  MoveL 3801 to (497.52, 492.57, 7.8) mm, rotated rx 0 ry 90 rz 0 deg; joints [-11.373, -27.183, 111.629, -15.362, -83.781, 50.697]
  MoveL 3802 to (497.65, 492.45, 7.8) mm, rotated rx 0 ry 90 rz 0 deg; joints [-11.359, -27.181, 111.617, -15.349, -83.771, 50.699]
  Set speed (120.0 mm/s)
  MoveL 3803 to (502.42, 492.52, 7.8) mm, rotated rx 0 ry 90 rz 0 deg; joints [-11.277, -27.097, 111.047, -15.281, -83.3, 50.82]
  Set speed (30.0 mm/s)
  Call Extruder(0.230)
  MoveL 3804 to (508, 498.1, 7.8) mm, rotated rx 0 ry 90 rz 0 deg; joints [-11.683, -26.971, 110.241, -15.712, -82.657, 51.047]
  MoveL 3805 to (508.13, 498.23, 7.8) mm, rotated rx 0 ry 90 rz 0 deg; joints [-11.692, -26.968, 110.224, -15.722, -82.643, 51.052]
  Set speed (120.0 mm/s)
  MoveL 3806 to (509.32, 490.68, 7.8) mm, rotated rx 0 ry 90 rz 0 deg; joints [-10.985, -26.974, 110.262, -15.009, -82.652, 50.963]
  Set speed (30.0 mm/s)
  Call Extruder(0.767)
  MoveL 3807 to (490.68, 509.32, 7.8) mm, rotated rx 0 ry 90 rz 0 deg; joints [-13.056, -27.238, 112.01, -17.045, -84.139, 50.759]
  MoveL 3808 to (490.56, 509.44, 7.8) mm, rotated rx 0 ry 90 rz 0 deg; joints [-13.07, -27.239, 112.021, -17.059, -84.148, 50.757]
  Set speed (120.0 mm/s)
  MoveL 3809 to (499.58, 492.37, 7.8) mm, rotated rx 0 ry 90 rz 0 deg; joints [-11.315, -27.148, 111.389, -15.311, -83.582, 50.746]
  Set speed (1000.0 mm/s)
  MoveL 3810 to (499.65, 492.3, 7.8) mm, rotated rx 0 ry 90 rz 0 deg; joints [-11.307, -27.147, 111.382, -15.303, -83.576, 50.747]
  Set speed (15.0 mm/s)
  Call Extruder(0.010)
  MoveL 3811 to (500, 492.3, 7.8) mm, rotated rx 0 ry 90 rz 0 deg; joints [-11.301, -27.141, 111.341, -15.297, -83.542, 50.756]
  Call Extruder(0.000)
  MoveL 3812 to (500, 492.3, 7.8) mm, rotated rx 0 ry 90 rz 0 deg; joints [-11.301, -27.141, 111.34, -15.297, -83.542, 50.756]
  Call Extruder(0.062)
  MoveL 3813 to (502.14, 492.3, 7.8) mm, rotated rx 0 ry 90 rz 0 deg; joints [-11.262, -27.102, 111.085, -15.265, -83.331, 50.81]
  Call Extruder(0.055)
  MoveL 3814 to (502.14, 490.4, 7.8) mm, rotated rx 0 ry 90 rz 0 deg; joints [-11.088, -27.109, 111.13, -15.088, -83.363, 50.782]
  Call Extruder(0.217)
  MoveL 3815 to (509.6, 490.4, 7.8) mm, rotated rx 0 ry 90 rz 0 deg; joints [-10.955, -26.97, 110.235, -14.979, -82.629, 50.965]
  Call Extruder(0.232)
  MoveL 3816 to (509.6, 498.38, 7.8) mm, rotated rx 0 ry 90 rz 0 deg; joints [-11.678, -26.939, 110.042, -15.714, -82.496, 51.092]
  Call Extruder(0.046)
  MoveL 3817 to (508.01, 498.39, 7.8) mm, rotated rx 0 ry 90 rz 0 deg; joints [-11.708, -26.97, 110.233, -15.738, -82.651, 51.051]
  Call Extruder(0.010)
  MoveL 3818 to (507.66, 498.38, 7.8) mm, rotated rx 0 ry 90 rz 0 deg; joints [-11.715, -26.977, 110.275, -15.743, -82.686, 51.043]
  Call Extruder(0.007)
  MoveL 3819 to (507.66, 498.74, 7.8) mm, rotated rx 0 ry 90 rz 0 deg; joints [-11.746, -26.975, 110.267, -15.776, -82.68, 51.048]
  Call Extruder(0.062)
  MoveL 3820 to (507.66, 500.87, 7.8) mm, rotated rx 0 ry 90 rz 0 deg; joints [-11.939, -26.967, 110.213, -15.971, -82.642, 51.083]
  Call Extruder(0.056)
  MoveL 3821 to (509.6, 500.87, 7.8) mm, rotated rx 0 ry 90 rz 0 deg; joints [-11.902, -26.929, 109.98, -15.941, -82.453, 51.132]
  Call Extruder(0.254)
  MoveL 3822 to (509.6, 509.6, 7.8) mm, rotated rx 0 ry 90 rz 0 deg; joints [-12.688, -26.891, 109.751, -16.741, -82.297, 51.28]
  Call Extruder(0.559)
  MoveL 3823 to (490.4, 509.6, 7.8) mm, rotated rx 0 ry 90 rz 0 deg; joints [-13.088, -27.241, 112.035, -17.076, -84.16, 50.755]
  MoveL 3824 to (490.4, 490.4, 7.8) mm, rotated rx 0 ry 90 rz 0 deg; joints [-11.303, -27.309, 112.525, -15.272, -84.522, 50.487]
  Call Extruder(0.189)
  MoveL 3825 to (496.9, 490.4, 7.8) mm, rotated rx 0 ry 90 rz 0 deg; joints [-11.183, -27.201, 111.755, -15.169, -83.88, 50.651]
  Call Extruder(0.055)
  MoveL 3826 to (496.9, 492.3, 7.8) mm, rotated rx 0 ry 90 rz 0 deg; joints [-11.358, -27.195, 111.71, -15.346, -83.847, 50.678]
  Call Extruder(0.075)
  MoveL 3827 to (499.46, 492.29, 7.8) mm, rotated rx 0 ry 90 rz 0 deg; joints [-11.311, -27.15, 111.405, -15.306, -83.595, 50.742]
  Call Extruder(0.021)
  MoveL 3828 to (499.46, 491.57, 7.8) mm, rotated rx 0 ry 90 rz 0 deg; joints [-11.244, -27.153, 111.422, -15.238, -83.607, 50.732]
  Call Extruder(0.034)
  MoveL 3829 to (499.46, 490.4, 7.8) mm, rotated rx 0 ry 90 rz 0 deg; joints [-11.136, -27.157, 111.45, -15.129, -83.627, 50.715]
  Call Extruder(0.006)
  MoveL 3830 to (499.66, 490.4, 7.8) mm, rotated rx 0 ry 90 rz 0 deg; joints [-11.133, -27.154, 111.427, -15.126, -83.608, 50.72]
  Call Extruder(0.009)
  MoveL 3831 to (499.66, 491.57, 7.8) mm, rotated rx 0 ry 90 rz 0 deg; joints [-11.241, -27.149, 111.399, -15.235, -83.588, 50.737]
  Call Extruder(0.011)
  MoveL 3832 to (499.65, 491.94, 7.8) mm, rotated rx 0 ry 90 rz 0 deg; joints [-11.275, -27.148, 111.391, -15.27, -83.582, 50.742]
  Call Extruder(0.000)
  MoveL 3833 to (499.65, 491.94, 7.8) mm, rotated rx 0 ry 90 rz 0 deg; joints [-11.275, -27.148, 111.391, -15.27, -83.582, 50.742]
  Call Extruder(0.007)
  MoveL 3834 to (499.65, 492.3, 7.8) mm, rotated rx 0 ry 90 rz 0 deg; joints [-11.307, -27.147, 111.382, -15.303, -83.576, 50.747]
  Set speed (120.0 mm/s)
  MoveL 3835 to (500, 492.3, 7.8) mm, rotated rx 0 ry 90 rz 0 deg; joints [-11.301, -27.141, 111.341, -15.297, -83.542, 50.756]
  Set speed (1000.0 mm/s)
  MoveL 3836 to (500, 492.3, 7.8) mm, rotated rx 0 ry 90 rz 0 deg; joints [-11.301, -27.141, 111.34, -15.297, -83.542, 50.756]
  Set speed (1000.0 mm/s)
  MoveL 3837 to (500.05, 492.3, 7.8) mm, rotated rx 0 ry 90 rz 0 deg; joints [-11.3, -27.14, 111.335, -15.297, -83.537, 50.757]
  Set speed (1000.0 mm/s)
  MoveL 3838 to (500.05, 493, 7.8) mm, rotated rx 0 ry 90 rz 0 deg; joints [-11.364, -27.137, 111.318, -15.362, -83.525, 50.767]
  Set speed (1000.0 mm/s)
  MoveL 3839 to (497.48, 492.45, 7.8) mm, rotated rx 0 ry 90 rz 0 deg; joints [-11.362, -27.184, 111.637, -15.352, -83.788, 50.695]
  Set speed (1000.0 mm/s)
  MoveL 3840 to (490.68, 490.68, 7.8) mm, rotated rx 0 ry 90 rz 0 deg; joints [-11.324, -27.303, 112.485, -15.294, -84.489, 50.498]
  Set speed (1000.0 mm/s)
  MoveL 3841 to (490.68, 490.68, 7.9) mm, rotated rx 0 ry 90 rz 0 deg; joints [-11.324, -27.314, 112.49, -15.294, -84.484, 50.499]
  Set speed (30.0 mm/s)
  Call Extruder(0.767)
  MoveL 3842 to (509.32, 509.32, 7.9) mm, rotated rx 0 ry 90 rz 0 deg; joints [-12.669, -26.909, 109.797, -16.72, -82.324, 51.269]
  MoveL 3843 to (509.44, 509.44, 7.9) mm, rotated rx 0 ry 90 rz 0 deg; joints [-12.677, -26.906, 109.779, -16.729, -82.31, 51.275]
  Set speed (120.0 mm/s)
  MoveL 3844 to (508.75, 501.14, 7.9) mm, rotated rx 0 ry 90 rz 0 deg; joints [-11.944, -26.955, 110.08, -15.98, -82.526, 51.117]
  Set speed (30.0 mm/s)
  Call Extruder(0.336)
  MoveL 3845 to (500.58, 509.32, 7.9) mm, rotated rx 0 ry 90 rz 0 deg; joints [-12.847, -27.075, 110.843, -16.868, -83.172, 51.033]
  Set speed (120.0 mm/s)
  MoveL 3846 to (499.42, 509.32, 7.9) mm, rotated rx 0 ry 90 rz 0 deg; joints [-12.872, -27.096, 110.981, -16.888, -83.284, 51.002]
  Set speed (30.0 mm/s)
  Call Extruder(0.360)
  MoveL 3847 to (490.68, 500.58, 7.9) mm, rotated rx 0 ry 90 rz 0 deg; joints [-12.247, -27.281, 112.247, -16.226, -84.303, 50.633]
  Set speed (120.0 mm/s)
  MoveL 3848 to (490.68, 499.42, 7.9) mm, rotated rx 0 ry 90 rz 0 deg; joints [-12.139, -27.285, 112.276, -16.117, -84.325, 50.617]
  Set speed (30.0 mm/s)
  Call Extruder(0.282)
  MoveL 3849 to (497.52, 492.58, 7.9) mm, rotated rx 0 ry 90 rz 0 deg; joints [-11.373, -27.194, 111.634, -15.362, -83.776, 50.699]
  MoveL 3850 to (497.65, 492.45, 7.9) mm, rotated rx 0 ry 90 rz 0 deg; joints [-11.359, -27.192, 111.623, -15.349, -83.766, 50.7]
  Set speed (120.0 mm/s)
  MoveL 3851 to (502.36, 492.46, 7.9) mm, rotated rx 0 ry 90 rz 0 deg; joints [-11.272, -27.109, 111.061, -15.276, -83.302, 50.819]
  Set speed (30.0 mm/s)
  Call Extruder(0.232)
  MoveL 3852 to (508, 498.1, 7.9) mm, rotated rx 0 ry 90 rz 0 deg; joints [-11.683, -26.982, 110.247, -15.712, -82.652, 51.048]
  MoveL 3853 to (508.13, 498.23, 7.9) mm, rotated rx 0 ry 90 rz 0 deg; joints [-11.692, -26.979, 110.229, -15.722, -82.638, 51.053]
  Set speed (120.0 mm/s)
  MoveL 3854 to (509.32, 490.68, 7.9) mm, rotated rx 0 ry 90 rz 0 deg; joints [-10.985, -26.985, 110.267, -15.009, -82.647, 50.964]
  Set speed (30.0 mm/s)
  Call Extruder(0.767)
  MoveL 3855 to (490.68, 509.32, 7.9) mm, rotated rx 0 ry 90 rz 0 deg; joints [-13.056, -27.248, 112.015, -17.045, -84.134, 50.76]
  MoveL 3856 to (490.56, 509.44, 7.9) mm, rotated rx 0 ry 90 rz 0 deg; joints [-13.07, -27.25, 112.027, -17.059, -84.143, 50.759]
  Set speed (120.0 mm/s)
  MoveL 3857 to (499.52, 492.37, 7.9) mm, rotated rx 0 ry 90 rz 0 deg; joints [-11.316, -27.16, 111.401, -15.312, -83.583, 50.746]
  Set speed (1000.0 mm/s)
  MoveL 3858 to (499.59, 492.29, 7.9) mm, rotated rx 0 ry 90 rz 0 deg; joints [-11.308, -27.159, 111.395, -15.304, -83.577, 50.747]
  Set speed (15.0 mm/s)
  Call Extruder(0.072)
  MoveL 3859 to (502.08, 492.3, 7.9) mm, rotated rx 0 ry 90 rz 0 deg; joints [-11.263, -27.114, 111.098, -15.266, -83.332, 50.809]
  Call Extruder(0.055)
  MoveL 3860 to (502.08, 490.4, 7.9) mm, rotated rx 0 ry 90 rz 0 deg; joints [-11.089, -27.121, 111.143, -15.089, -83.364, 50.782]
  Call Extruder(0.219)
  MoveL 3861 to (509.6, 490.4, 7.9) mm, rotated rx 0 ry 90 rz 0 deg; joints [-10.955, -26.981, 110.24, -14.979, -82.624, 50.967]
  Call Extruder(0.232)
  MoveL 3862 to (509.6, 498.38, 7.9) mm, rotated rx 0 ry 90 rz 0 deg; joints [-11.678, -26.95, 110.048, -15.714, -82.491, 51.093]
  Call Extruder(0.046)
  MoveL 3863 to (508.01, 498.38, 7.9) mm, rotated rx 0 ry 90 rz 0 deg; joints [-11.708, -26.98, 110.239, -15.738, -82.646, 51.053]
  Call Extruder(0.010)
  MoveL 3864 to (507.66, 498.38, 7.9) mm, rotated rx 0 ry 90 rz 0 deg; joints [-11.715, -26.987, 110.281, -15.743, -82.681, 51.044]
  Call Extruder(0.007)
  MoveL 3865 to (507.66, 498.73, 7.9) mm, rotated rx 0 ry 90 rz 0 deg; joints [-11.746, -26.986, 110.272, -15.776, -82.675, 51.05]
  Call Extruder(0.062)
  MoveL 3866 to (507.66, 500.86, 7.9) mm, rotated rx 0 ry 90 rz 0 deg; joints [-11.939, -26.977, 110.218, -15.971, -82.637, 51.084]
  Call Extruder(0.056)
  MoveL 3867 to (509.6, 500.87, 7.9) mm, rotated rx 0 ry 90 rz 0 deg; joints [-11.902, -26.939, 109.985, -15.942, -82.448, 51.134]
  Call Extruder(0.254)
  MoveL 3868 to (509.6, 509.6, 7.9) mm, rotated rx 0 ry 90 rz 0 deg; joints [-12.688, -26.902, 109.756, -16.741, -82.292, 51.282]
  Call Extruder(0.559)
  MoveL 3869 to (490.4, 509.6, 7.9) mm, rotated rx 0 ry 90 rz 0 deg; joints [-13.088, -27.252, 112.041, -17.076, -84.155, 50.757]
  MoveL 3870 to (490.4, 490.4, 7.9) mm, rotated rx 0 ry 90 rz 0 deg; joints [-11.303, -27.319, 112.53, -15.272, -84.517, 50.488]
  Call Extruder(0.191)
  MoveL 3871 to (496.95, 490.4, 7.9) mm, rotated rx 0 ry 90 rz 0 deg; joints [-11.182, -27.211, 111.753, -15.168, -83.869, 50.654]
  Call Extruder(0.055)
  MoveL 3872 to (496.96, 492.3, 7.9) mm, rotated rx 0 ry 90 rz 0 deg; joints [-11.357, -27.204, 111.708, -15.345, -83.836, 50.681]
  Call Extruder(0.074)
  MoveL 3873 to (499.51, 492.29, 7.9) mm, rotated rx 0 ry 90 rz 0 deg; joints [-11.31, -27.16, 111.404, -15.305, -83.585, 50.745]
  Call Extruder(0.000)
  MoveL 3874 to (499.52, 492.29, 7.9) mm, rotated rx 0 ry 90 rz 0 deg; joints [-11.31, -27.16, 111.403, -15.305, -83.584, 50.745]
  Call Extruder(0.020)
  MoveL 3875 to (499.52, 491.61, 7.9) mm, rotated rx 0 ry 90 rz 0 deg; joints [-11.247, -27.162, 111.419, -15.242, -83.595, 50.736]
  Call Extruder(0.000)
  MoveL 3876 to (499.52, 491.6, 7.9) mm, rotated rx 0 ry 90 rz 0 deg; joints [-11.246, -27.162, 111.419, -15.241, -83.595, 50.735]
  Call Extruder(0.000)
  MoveL 3877 to (499.52, 491.6, 7.9) mm, rotated rx 0 ry 90 rz 0 deg; joints [-11.246, -27.162, 111.419, -15.241, -83.595, 50.735]
  Call Extruder(0.035)
  MoveL 3878 to (499.52, 490.4, 7.9) mm, rotated rx 0 ry 90 rz 0 deg; joints [-11.135, -27.166, 111.448, -15.128, -83.616, 50.718]
  Call Extruder(0.002)
  MoveL 3879 to (499.59, 490.4, 7.9) mm, rotated rx 0 ry 90 rz 0 deg; joints [-11.134, -27.165, 111.439, -15.127, -83.609, 50.72]
  Call Extruder(0.019)
  MoveL 3880 to (499.59, 491.6, 7.9) mm, rotated rx 0 ry 90 rz 0 deg; joints [-11.245, -27.161, 111.411, -15.24, -83.589, 50.737]
  Call Extruder(0.000)
  MoveL 3881 to (499.6, 491.61, 7.9) mm, rotated rx 0 ry 90 rz 0 deg; joints [-11.245, -27.161, 111.411, -15.24, -83.588, 50.737]
  Call Extruder(0.002)
  MoveL 3882 to (499.59, 492.29, 7.9) mm, rotated rx 0 ry 90 rz 0 deg; joints [-11.308, -27.159, 111.395, -15.304, -83.577, 50.747]
  Set speed (120.0 mm/s)
  MoveL 3883 to (499.99, 492.3, 7.9) mm, rotated rx 0 ry 90 rz 0 deg; joints [-11.301, -27.151, 111.347, -15.298, -83.538, 50.757]
  Set speed (1000.0 mm/s)
  MoveL 3884 to (499.99, 492.99, 7.9) mm, rotated rx 0 ry 90 rz 0 deg; joints [-11.365, -27.149, 111.33, -15.363, -83.525, 50.767]
  Set speed (1000.0 mm/s)
  MoveL 3885 to (497.51, 492.45, 7.9) mm, rotated rx 0 ry 90 rz 0 deg; joints [-11.361, -27.194, 111.639, -15.351, -83.779, 50.697]
  Set speed (1000.0 mm/s)
  MoveL 3886 to (490.68, 490.68, 7.9) mm, rotated rx 0 ry 90 rz 0 deg; joints [-11.324, -27.314, 112.49, -15.294, -84.484, 50.499]
  Set speed (1000.0 mm/s)
  MoveL 3887 to (490.68, 490.68, 8) mm, rotated rx 0 ry 90 rz 0 deg; joints [-11.324, -27.325, 112.496, -15.294, -84.479, 50.501]
  Set speed (30.0 mm/s)
  Call Extruder(0.767)
  MoveL 3888 to (509.32, 509.32, 8) mm, rotated rx 0 ry 90 rz 0 deg; joints [-12.669, -26.919, 109.803, -16.72, -82.319, 51.271]
  MoveL 3889 to (509.44, 509.44, 8) mm, rotated rx 0 ry 90 rz 0 deg; joints [-12.677, -26.916, 109.785, -16.729, -82.305, 51.276]
  Set speed (120.0 mm/s)
  MoveL 3890 to (508.75, 501.14, 8) mm, rotated rx 0 ry 90 rz 0 deg; joints [-11.944, -26.965, 110.085, -15.98, -82.521, 51.118]
  Set speed (30.0 mm/s)
  Call Extruder(0.337)
  MoveL 3891 to (500.58, 509.32, 8) mm, rotated rx 0 ry 90 rz 0 deg; joints [-12.847, -27.086, 110.849, -16.868, -83.167, 51.035]
  Set speed (120.0 mm/s)
  MoveL 3892 to (499.42, 509.32, 8) mm, rotated rx 0 ry 90 rz 0 deg; joints [-12.872, -27.107, 110.986, -16.888, -83.279, 51.003]
  Set speed (30.0 mm/s)
  Call Extruder(0.360)
  MoveL 3893 to (490.68, 500.58, 8) mm, rotated rx 0 ry 90 rz 0 deg; joints [-12.247, -27.291, 112.252, -16.226, -84.298, 50.635]
  Set speed (120.0 mm/s)
  MoveL 3894 to (490.68, 499.42, 8) mm, rotated rx 0 ry 90 rz 0 deg; joints [-12.139, -27.295, 112.282, -16.117, -84.32, 50.618]
  Set speed (30.0 mm/s)
  Call Extruder(0.282)
  MoveL 3895 to (497.52, 492.58, 8) mm, rotated rx 0 ry 90 rz 0 deg; joints [-11.373, -27.204, 111.64, -15.363, -83.771, 50.7]
  MoveL 3896 to (497.65, 492.45, 8) mm, rotated rx 0 ry 90 rz 0 deg; joints [-11.359, -27.203, 111.628, -15.349, -83.761, 50.702]
  Set speed (120.0 mm/s)
  MoveL 3897 to (502.29, 492.39, 8) mm, rotated rx 0 ry 90 rz 0 deg; joints [-11.268, -27.121, 111.075, -15.272, -83.304, 50.818]
  Set speed (30.0 mm/s)
  Call Extruder(0.235)
  MoveL 3898 to (508, 498.1, 8) mm, rotated rx 0 ry 90 rz 0 deg; joints [-11.683, -26.992, 110.252, -15.712, -82.647, 51.05]
  MoveL 3899 to (508.13, 498.23, 8) mm, rotated rx 0 ry 90 rz 0 deg; joints [-11.692, -26.989, 110.234, -15.722, -82.633, 51.055]
  Set speed (120.0 mm/s)
  MoveL 3900 to (509.32, 490.68, 8) mm, rotated rx 0 ry 90 rz 0 deg; joints [-10.985, -26.995, 110.273, -15.009, -82.642, 50.965]
  Set speed (30.0 mm/s)
  Call Extruder(0.767)
  MoveL 3901 to (490.68, 509.32, 8) mm, rotated rx 0 ry 90 rz 0 deg; joints [-13.056, -27.259, 112.021, -17.045, -84.128, 50.762]
  MoveL 3902 to (490.56, 509.44, 8) mm, rotated rx 0 ry 90 rz 0 deg; joints [-13.07, -27.261, 112.032, -17.059, -84.138, 50.76]
  Set speed (120.0 mm/s)
  MoveL 3903 to (507.59, 498.31, 8) mm, rotated rx 0 ry 90 rz 0 deg; joints [-11.71, -26.999, 110.296, -15.738, -82.684, 51.043]
  Set speed (1000.0 mm/s)
  MoveL 3904 to (507.66, 498.38, 8) mm, rotated rx 0 ry 90 rz 0 deg; joints [-11.715, -26.998, 110.286, -15.743, -82.676, 51.045]
  Set speed (15.0 mm/s)
  Call Extruder(0.049)
  MoveL 3905 to (507.66, 500.07, 8) mm, rotated rx 0 ry 90 rz 0 deg; joints [-11.868, -26.991, 110.244, -15.899, -82.646, 51.073]
  Call Extruder(0.023)
  MoveL 3906 to (507.66, 500.86, 8) mm, rotated rx 0 ry 90 rz 0 deg; joints [-11.939, -26.988, 110.224, -15.972, -82.632, 51.085]
  Call Extruder(0.056)
  MoveL 3907 to (509.6, 500.87, 8) mm, rotated rx 0 ry 90 rz 0 deg; joints [-11.902, -26.95, 109.99, -15.942, -82.443, 51.135]
  Call Extruder(0.254)
  MoveL 3908 to (509.6, 509.6, 8) mm, rotated rx 0 ry 90 rz 0 deg; joints [-12.688, -26.912, 109.761, -16.741, -82.287, 51.283]
  Call Extruder(0.559)
  MoveL 3909 to (490.4, 509.6, 8) mm, rotated rx 0 ry 90 rz 0 deg; joints [-13.088, -27.263, 112.046, -17.077, -84.15, 50.758]
  MoveL 3910 to (490.4, 490.4, 8) mm, rotated rx 0 ry 90 rz 0 deg; joints [-11.303, -27.33, 112.535, -15.272, -84.511, 50.49]
  Call Extruder(0.192)
  MoveL 3911 to (497.01, 490.4, 8) mm, rotated rx 0 ry 90 rz 0 deg; joints [-11.181, -27.221, 111.752, -15.167, -83.859, 50.657]
  Call Extruder(0.055)
  MoveL 3912 to (497.01, 492.3, 8) mm, rotated rx 0 ry 90 rz 0 deg; joints [-11.356, -27.214, 111.707, -15.345, -83.826, 50.683]
  Call Extruder(0.146)
  MoveL 3913 to (502.02, 492.3, 8) mm, rotated rx 0 ry 90 rz 0 deg; joints [-11.264, -27.126, 111.111, -15.267, -83.333, 50.809]
  Call Extruder(0.055)
  MoveL 3914 to (502.02, 490.4, 8) mm, rotated rx 0 ry 90 rz 0 deg; joints [-11.09, -27.133, 111.155, -15.091, -83.365, 50.782]
  Call Extruder(0.221)
  MoveL 3915 to (509.6, 490.4, 8) mm, rotated rx 0 ry 90 rz 0 deg; joints [-10.955, -26.991, 110.245, -14.979, -82.619, 50.968]
  Call Extruder(0.232)
  MoveL 3916 to (509.6, 498.38, 8) mm, rotated rx 0 ry 90 rz 0 deg; joints [-11.678, -26.96, 110.053, -15.714, -82.486, 51.095]
  Call Extruder(0.056)
  MoveL 3917 to (507.66, 498.38, 8) mm, rotated rx 0 ry 90 rz 0 deg; joints [-11.715, -26.998, 110.286, -15.743, -82.676, 51.045]
  Set speed (120.0 mm/s)
  MoveL 3918 to (507.66, 498.78, 8) mm, rotated rx 0 ry 90 rz 0 deg; joints [-11.751, -26.996, 110.276, -15.78, -82.669, 51.052]
  Set speed (1000.0 mm/s)
  MoveL 3919 to (506.96, 498.78, 8) mm, rotated rx 0 ry 90 rz 0 deg; joints [-11.764, -27.009, 110.36, -15.791, -82.737, 51.034]
  Set speed (1000.0 mm/s)
  MoveL 3920 to (490.68, 490.68, 8) mm, rotated rx 0 ry 90 rz 0 deg; joints [-11.324, -27.325, 112.496, -15.294, -84.479, 50.501]
  Set speed (1000.0 mm/s)
  MoveL 3921 to (490.68, 490.68, 8.1) mm, rotated rx 0 ry 90 rz 0 deg; joints [-11.324, -27.335, 112.501, -15.294, -84.474, 50.502]
  Set speed (30.0 mm/s)
  Call Extruder(0.767)
  MoveL 3922 to (509.32, 509.32, 8.1) mm, rotated rx 0 ry 90 rz 0 deg; joints [-12.669, -26.93, 109.808, -16.72, -82.314, 51.272]
  MoveL 3923 to (509.44, 509.44, 8.1) mm, rotated rx 0 ry 90 rz 0 deg; joints [-12.677, -26.927, 109.79, -16.73, -82.3, 51.278]
  Set speed (120.0 mm/s)
  MoveL 3924 to (508.76, 501.14, 8.1) mm, rotated rx 0 ry 90 rz 0 deg; joints [-11.943, -26.976, 110.09, -15.98, -82.516, 51.12]
  Set speed (30.0 mm/s)
  Call Extruder(0.337)
  MoveL 3925 to (500.58, 509.32, 8.1) mm, rotated rx 0 ry 90 rz 0 deg; joints [-12.847, -27.096, 110.854, -16.868, -83.162, 51.036]
  Set speed (120.0 mm/s)
  MoveL 3926 to (499.42, 509.32, 8.1) mm, rotated rx 0 ry 90 rz 0 deg; joints [-12.872, -27.118, 110.992, -16.888, -83.274, 51.005]
  Set speed (30.0 mm/s)
  Call Extruder(0.360)
  MoveL 3927 to (490.68, 500.58, 8.1) mm, rotated rx 0 ry 90 rz 0 deg; joints [-12.247, -27.302, 112.257, -16.226, -84.293, 50.636]
  Set speed (120.0 mm/s)
  MoveL 3928 to (490.68, 499.42, 8.1) mm, rotated rx 0 ry 90 rz 0 deg; joints [-12.139, -27.306, 112.287, -16.117, -84.315, 50.62]
  Set speed (30.0 mm/s)
  Call Extruder(0.282)
  MoveL 3929 to (497.52, 492.57, 8.1) mm, rotated rx 0 ry 90 rz 0 deg; joints [-11.373, -27.215, 111.645, -15.363, -83.766, 50.702]
  MoveL 3930 to (497.65, 492.45, 8.1) mm, rotated rx 0 ry 90 rz 0 deg; joints [-11.359, -27.213, 111.633, -15.349, -83.756, 50.703]
  Set speed (120.0 mm/s)
  MoveL 3931 to (502.23, 492.33, 8.1) mm, rotated rx 0 ry 90 rz 0 deg; joints [-11.263, -27.132, 111.09, -15.267, -83.307, 50.817]
  Set speed (30.0 mm/s)
  Call Extruder(0.238)
  MoveL 3932 to (508, 498.1, 8.1) mm, rotated rx 0 ry 90 rz 0 deg; joints [-11.683, -27.003, 110.257, -15.712, -82.642, 51.051]
  MoveL 3933 to (508.12, 498.22, 8.1) mm, rotated rx 0 ry 90 rz 0 deg; joints [-11.691, -27, 110.24, -15.722, -82.628, 51.056]
  Set speed (120.0 mm/s)
  MoveL 3934 to (509.32, 490.68, 8.1) mm, rotated rx 0 ry 90 rz 0 deg; joints [-10.985, -27.006, 110.278, -15.009, -82.637, 50.967]
  Set speed (30.0 mm/s)
  Call Extruder(0.767)
  MoveL 3935 to (490.68, 509.32, 8.1) mm, rotated rx 0 ry 90 rz 0 deg; joints [-13.056, -27.27, 112.026, -17.045, -84.123, 50.763]
  MoveL 3936 to (490.56, 509.44, 8.1) mm, rotated rx 0 ry 90 rz 0 deg; joints [-13.07, -27.271, 112.037, -17.059, -84.133, 50.762]
  Set speed (120.0 mm/s)
  MoveL 3937 to (507.59, 498.31, 8.1) mm, rotated rx 0 ry 90 rz 0 deg; joints [-11.709, -27.01, 110.301, -15.738, -82.679, 51.044]
  Set speed (1000.0 mm/s)
  MoveL 3938 to (507.66, 498.38, 8.1) mm, rotated rx 0 ry 90 rz 0 deg; joints [-11.714, -27.008, 110.291, -15.744, -82.671, 51.047]
  Set speed (15.0 mm/s)
  Call Extruder(0.072)
  MoveL 3939 to (507.66, 500.86, 8.1) mm, rotated rx 0 ry 90 rz 0 deg; joints [-11.939, -26.998, 110.229, -15.972, -82.627, 51.087]
  Call Extruder(0.056)
  MoveL 3940 to (509.6, 500.86, 8.1) mm, rotated rx 0 ry 90 rz 0 deg; joints [-11.902, -26.96, 109.996, -15.942, -82.438, 51.137]
  Call Extruder(0.254)
  MoveL 3941 to (509.6, 509.6, 8.1) mm, rotated rx 0 ry 90 rz 0 deg; joints [-12.688, -26.923, 109.767, -16.741, -82.282, 51.285]
  Call Extruder(0.559)
  MoveL 3942 to (490.4, 509.6, 8.1) mm, rotated rx 0 ry 90 rz 0 deg; joints [-13.088, -27.273, 112.051, -17.077, -84.145, 50.76]
  MoveL 3943 to (490.4, 490.4, 8.1) mm, rotated rx 0 ry 90 rz 0 deg; joints [-11.303, -27.341, 112.541, -15.272, -84.506, 50.491]
  Call Extruder(0.194)
  MoveL 3944 to (497.07, 490.4, 8.1) mm, rotated rx 0 ry 90 rz 0 deg; joints [-11.18, -27.23, 111.751, -15.166, -83.848, 50.66]
  Call Extruder(0.055)
  MoveL 3945 to (497.07, 492.3, 8.1) mm, rotated rx 0 ry 90 rz 0 deg; joints [-11.355, -27.224, 111.706, -15.344, -83.815, 50.686]
  Call Extruder(0.142)
  MoveL 3946 to (501.95, 492.3, 8.1) mm, rotated rx 0 ry 90 rz 0 deg; joints [-11.265, -27.138, 111.124, -15.268, -83.335, 50.809]
  Call Extruder(0.055)
  MoveL 3947 to (501.95, 490.4, 8.1) mm, rotated rx 0 ry 90 rz 0 deg; joints [-11.091, -27.144, 111.168, -15.092, -83.366, 50.782]
  Call Extruder(0.223)
  MoveL 3948 to (509.6, 490.4, 8.1) mm, rotated rx 0 ry 90 rz 0 deg; joints [-10.955, -27.002, 110.25, -14.979, -82.614, 50.969]
  Call Extruder(0.232)
  MoveL 3949 to (509.6, 498.38, 8.1) mm, rotated rx 0 ry 90 rz 0 deg; joints [-11.678, -26.97, 110.058, -15.714, -82.481, 51.096]
  Call Extruder(0.056)
  MoveL 3950 to (507.66, 498.38, 8.1) mm, rotated rx 0 ry 90 rz 0 deg; joints [-11.714, -27.008, 110.291, -15.744, -82.671, 51.047]
  Set speed (120.0 mm/s)
  MoveL 3951 to (507.66, 498.78, 8.1) mm, rotated rx 0 ry 90 rz 0 deg; joints [-11.751, -27.006, 110.281, -15.78, -82.664, 51.053]
  Set speed (1000.0 mm/s)
  MoveL 3952 to (506.96, 498.78, 8.1) mm, rotated rx 0 ry 90 rz 0 deg; joints [-11.764, -27.02, 110.365, -15.791, -82.732, 51.035]
  Set speed (1000.0 mm/s)
  MoveL 3953 to (490.68, 490.68, 8.1) mm, rotated rx 0 ry 90 rz 0 deg; joints [-11.324, -27.335, 112.501, -15.294, -84.474, 50.502]
  Set speed (1000.0 mm/s)
  MoveL 3954 to (490.68, 490.68, 8.2) mm, rotated rx 0 ry 90 rz 0 deg; joints [-11.324, -27.346, 112.506, -15.294, -84.469, 50.503]
  Set speed (30.0 mm/s)
  Call Extruder(0.767)
  MoveL 3955 to (509.32, 509.32, 8.2) mm, rotated rx 0 ry 90 rz 0 deg; joints [-12.669, -26.94, 109.813, -16.721, -82.309, 51.274]
  MoveL 3956 to (509.44, 509.44, 8.2) mm, rotated rx 0 ry 90 rz 0 deg; joints [-12.677, -26.937, 109.795, -16.73, -82.295, 51.279]
  Set speed (120.0 mm/s)
  MoveL 3957 to (508.76, 501.14, 8.2) mm, rotated rx 0 ry 90 rz 0 deg; joints [-11.943, -26.986, 110.095, -15.98, -82.511, 51.121]
  Set speed (30.0 mm/s)
  Call Extruder(0.337)
  MoveL 3958 to (500.58, 509.32, 8.2) mm, rotated rx 0 ry 90 rz 0 deg; joints [-12.847, -27.107, 110.859, -16.868, -83.156, 51.038]
  Set speed (120.0 mm/s)
  MoveL 3959 to (499.42, 509.32, 8.2) mm, rotated rx 0 ry 90 rz 0 deg; joints [-12.872, -27.128, 110.997, -16.888, -83.269, 51.006]
  Set speed (30.0 mm/s)
  Call Extruder(0.360)
  MoveL 3960 to (490.68, 500.58, 8.2) mm, rotated rx 0 ry 90 rz 0 deg; joints [-12.247, -27.313, 112.263, -16.227, -84.288, 50.638]
  Set speed (120.0 mm/s)
  MoveL 3961 to (490.68, 499.42, 8.2) mm, rotated rx 0 ry 90 rz 0 deg; joints [-12.139, -27.317, 112.292, -16.118, -84.31, 50.621]
  Set speed (30.0 mm/s)
  Call Extruder(0.282)
  MoveL 3962 to (497.52, 492.58, 8.2) mm, rotated rx 0 ry 90 rz 0 deg; joints [-11.373, -27.226, 111.65, -15.363, -83.76, 50.703]
  MoveL 3963 to (497.65, 492.45, 8.2) mm, rotated rx 0 ry 90 rz 0 deg; joints [-11.359, -27.224, 111.638, -15.35, -83.75, 50.704]
  Set speed (120.0 mm/s)
  MoveL 3964 to (501.92, 492.32, 8.2) mm, rotated rx 0 ry 90 rz 0 deg; joints [-11.268, -27.149, 111.132, -15.271, -83.332, 50.81]
  Set speed (1000.0 mm/s)
  MoveL 3965 to (502.17, 492.27, 8.2) mm, rotated rx 0 ry 90 rz 0 deg; joints [-11.259, -27.144, 111.104, -15.262, -83.309, 50.816]
  Set speed (30.0 mm/s)
  Call Extruder(0.240)
  MoveL 3966 to (508, 498.1, 8.2) mm, rotated rx 0 ry 90 rz 0 deg; joints [-11.683, -27.013, 110.263, -15.713, -82.637, 51.052]
  MoveL 3967 to (508.12, 498.22, 8.2) mm, rotated rx 0 ry 90 rz 0 deg; joints [-11.691, -27.01, 110.245, -15.722, -82.623, 51.057]
  Set speed (120.0 mm/s)
  MoveL 3968 to (509.32, 490.68, 8.2) mm, rotated rx 0 ry 90 rz 0 deg; joints [-10.985, -27.016, 110.283, -15.009, -82.632, 50.968]
  Set speed (30.0 mm/s)
  Call Extruder(0.767)
  MoveL 3969 to (490.68, 509.32, 8.2) mm, rotated rx 0 ry 90 rz 0 deg; joints [-13.056, -27.28, 112.031, -17.046, -84.118, 50.765]
  MoveL 3970 to (490.56, 509.44, 8.2) mm, rotated rx 0 ry 90 rz 0 deg; joints [-13.07, -27.282, 112.042, -17.059, -84.128, 50.763]
  Set speed (120.0 mm/s)
  MoveL 3971 to (507.59, 498.31, 8.2) mm, rotated rx 0 ry 90 rz 0 deg; joints [-11.709, -27.02, 110.307, -15.738, -82.674, 51.045]
  Set speed (1000.0 mm/s)
  MoveL 3972 to (507.66, 498.38, 8.2) mm, rotated rx 0 ry 90 rz 0 deg; joints [-11.714, -27.019, 110.297, -15.744, -82.666, 51.048]
  Set speed (15.0 mm/s)
  Call Extruder(0.072)
  MoveL 3973 to (507.66, 500.86, 8.2) mm, rotated rx 0 ry 90 rz 0 deg; joints [-11.939, -27.009, 110.234, -15.972, -82.622, 51.088]
  Call Extruder(0.056)
  MoveL 3974 to (509.6, 500.86, 8.2) mm, rotated rx 0 ry 90 rz 0 deg; joints [-11.902, -26.971, 110.001, -15.942, -82.433, 51.138]
  Call Extruder(0.254)
  MoveL 3975 to (509.6, 509.6, 8.2) mm, rotated rx 0 ry 90 rz 0 deg; joints [-12.688, -26.933, 109.772, -16.742, -82.277, 51.286]
  Call Extruder(0.559)
  MoveL 3976 to (490.4, 509.6, 8.2) mm, rotated rx 0 ry 90 rz 0 deg; joints [-13.088, -27.284, 112.056, -17.077, -84.14, 50.761]
  MoveL 3977 to (490.4, 490.4, 8.2) mm, rotated rx 0 ry 90 rz 0 deg; joints [-11.303, -27.351, 112.546, -15.272, -84.501, 50.493]
  Call Extruder(0.196)
  MoveL 3978 to (497.12, 490.4, 8.2) mm, rotated rx 0 ry 90 rz 0 deg; joints [-11.179, -27.24, 111.749, -15.166, -83.837, 50.662]
  Call Extruder(0.055)
  MoveL 3979 to (497.12, 492.3, 8.2) mm, rotated rx 0 ry 90 rz 0 deg; joints [-11.354, -27.233, 111.704, -15.343, -83.805, 50.689]
  Call Extruder(0.139)
  MoveL 3980 to (501.89, 492.3, 8.2) mm, rotated rx 0 ry 90 rz 0 deg; joints [-11.266, -27.149, 111.136, -15.269, -83.336, 50.809]
  Call Extruder(0.055)
  MoveL 3981 to (501.89, 490.4, 8.2) mm, rotated rx 0 ry 90 rz 0 deg; joints [-11.092, -27.156, 111.181, -15.093, -83.367, 50.781]
  Call Extruder(0.224)
  MoveL 3982 to (509.6, 490.4, 8.2) mm, rotated rx 0 ry 90 rz 0 deg; joints [-10.955, -27.012, 110.256, -14.979, -82.609, 50.971]
  Call Extruder(0.232)
  MoveL 3983 to (509.6, 498.38, 8.2) mm, rotated rx 0 ry 90 rz 0 deg; joints [-11.678, -26.981, 110.063, -15.714, -82.476, 51.098]
  Call Extruder(0.056)
  MoveL 3984 to (507.66, 498.38, 8.2) mm, rotated rx 0 ry 90 rz 0 deg; joints [-11.714, -27.019, 110.297, -15.744, -82.666, 51.048]
  Set speed (120.0 mm/s)
  MoveL 3985 to (507.66, 498.78, 8.2) mm, rotated rx 0 ry 90 rz 0 deg; joints [-11.751, -27.017, 110.287, -15.78, -82.659, 51.055]
  Set speed (1000.0 mm/s)
  MoveL 3986 to (506.96, 498.78, 8.2) mm, rotated rx 0 ry 90 rz 0 deg; joints [-11.764, -27.03, 110.371, -15.791, -82.727, 51.037]
  Set speed (1000.0 mm/s)
  MoveL 3987 to (490.68, 490.68, 8.2) mm, rotated rx 0 ry 90 rz 0 deg; joints [-11.324, -27.346, 112.506, -15.294, -84.469, 50.503]
  Set speed (1000.0 mm/s)
  MoveL 3988 to (490.68, 490.68, 8.3) mm, rotated rx 0 ry 90 rz 0 deg; joints [-11.324, -27.357, 112.512, -15.294, -84.463, 50.505]
  Set speed (30.0 mm/s)
  Call Extruder(0.767)
  MoveL 3989 to (509.32, 509.32, 8.3) mm, rotated rx 0 ry 90 rz 0 deg; joints [-12.669, -26.95, 109.818, -16.721, -82.304, 51.275]
  MoveL 3990 to (509.44, 509.44, 8.3) mm, rotated rx 0 ry 90 rz 0 deg; joints [-12.677, -26.947, 109.8, -16.73, -82.29, 51.281]
  Set speed (120.0 mm/s)
  MoveL 3991 to (508.76, 501.14, 8.3) mm, rotated rx 0 ry 90 rz 0 deg; joints [-11.943, -26.997, 110.1, -15.981, -82.505, 51.123]
  Set speed (30.0 mm/s)
  Call Extruder(0.337)
  MoveL 3992 to (500.58, 509.32, 8.3) mm, rotated rx 0 ry 90 rz 0 deg; joints [-12.847, -27.117, 110.864, -16.868, -83.151, 51.039]
  Set speed (120.0 mm/s)
  MoveL 3993 to (499.42, 509.32, 8.3) mm, rotated rx 0 ry 90 rz 0 deg; joints [-12.872, -27.139, 111.002, -16.889, -83.264, 51.008]
  Set speed (30.0 mm/s)
  Call Extruder(0.360)
  MoveL 3994 to (490.68, 500.58, 8.3) mm, rotated rx 0 ry 90 rz 0 deg; joints [-12.247, -27.323, 112.268, -16.227, -84.283, 50.639]
  Set speed (120.0 mm/s)
  MoveL 3995 to (490.68, 499.42, 8.3) mm, rotated rx 0 ry 90 rz 0 deg; joints [-12.139, -27.327, 112.297, -16.118, -84.305, 50.623]
  Set speed (30.0 mm/s)
  Call Extruder(0.282)
  MoveL 3996 to (497.52, 492.58, 8.3) mm, rotated rx 0 ry 90 rz 0 deg; joints [-11.373, -27.236, 111.655, -15.363, -83.755, 50.705]
  MoveL 3997 to (497.65, 492.45, 8.3) mm, rotated rx 0 ry 90 rz 0 deg; joints [-11.359, -27.234, 111.644, -15.35, -83.745, 50.706]
  Set speed (120.0 mm/s)
  MoveL 3998 to (501.85, 492.32, 8.3) mm, rotated rx 0 ry 90 rz 0 deg; joints [-11.27, -27.16, 111.145, -15.273, -83.334, 50.81]
  Set speed (1000.0 mm/s)
  MoveL 3999 to (502.1, 492.2, 8.3) mm, rotated rx 0 ry 90 rz 0 deg; joints [-11.254, -27.156, 111.118, -15.257, -83.311, 50.814]
  Set speed (30.0 mm/s)
  Call Extruder(0.243)
  MoveL 4000 to (508, 498.1, 8.3) mm, rotated rx 0 ry 90 rz 0 deg; joints [-11.682, -27.024, 110.268, -15.713, -82.632, 51.054]
  MoveL 4001 to (508.12, 498.22, 8.3) mm, rotated rx 0 ry 90 rz 0 deg; joints [-11.691, -27.021, 110.25, -15.722, -82.618, 51.059]
  Set speed (120.0 mm/s)
  MoveL 4002 to (509.32, 490.68, 8.3) mm, rotated rx 0 ry 90 rz 0 deg; joints [-10.985, -27.027, 110.288, -15.009, -82.627, 50.97]
  Set speed (30.0 mm/s)
  Call Extruder(0.767)
  MoveL 4003 to (490.68, 509.32, 8.3) mm, rotated rx 0 ry 90 rz 0 deg; joints [-13.056, -27.291, 112.037, -17.046, -84.113, 50.766]
  MoveL 4004 to (490.56, 509.44, 8.3) mm, rotated rx 0 ry 90 rz 0 deg; joints [-13.07, -27.292, 112.048, -17.059, -84.123, 50.765]
  Set speed (120.0 mm/s)
  MoveL 4005 to (507.59, 498.31, 8.3) mm, rotated rx 0 ry 90 rz 0 deg; joints [-11.709, -27.031, 110.312, -15.738, -82.668, 51.047]
  Set speed (1000.0 mm/s)
  MoveL 4006 to (507.66, 498.38, 8.3) mm, rotated rx 0 ry 90 rz 0 deg; joints [-11.714, -27.029, 110.302, -15.744, -82.66, 51.05]
  Set speed (15.0 mm/s)
  Call Extruder(0.072)
  MoveL 4007 to (507.66, 500.86, 8.3) mm, rotated rx 0 ry 90 rz 0 deg; joints [-11.939, -27.019, 110.239, -15.972, -82.617, 51.09]
  Call Extruder(0.056)
  MoveL 4008 to (509.6, 500.86, 8.3) mm, rotated rx 0 ry 90 rz 0 deg; joints [-11.902, -26.981, 110.006, -15.942, -82.428, 51.14]
  Call Extruder(0.254)
  MoveL 4009 to (509.6, 509.6, 8.3) mm, rotated rx 0 ry 90 rz 0 deg; joints [-12.688, -26.944, 109.777, -16.742, -82.272, 51.288]
  Call Extruder(0.559)
  MoveL 4010 to (490.4, 509.6, 8.3) mm, rotated rx 0 ry 90 rz 0 deg; joints [-13.088, -27.294, 112.062, -17.077, -84.135, 50.763]
  MoveL 4011 to (490.4, 490.4, 8.3) mm, rotated rx 0 ry 90 rz 0 deg; joints [-11.303, -27.362, 112.551, -15.272, -84.496, 50.494]
  Call Extruder(0.197)
  MoveL 4012 to (497.18, 490.4, 8.3) mm, rotated rx 0 ry 90 rz 0 deg; joints [-11.178, -27.25, 111.748, -15.165, -83.827, 50.665]
  Call Extruder(0.055)
  MoveL 4013 to (497.18, 492.3, 8.3) mm, rotated rx 0 ry 90 rz 0 deg; joints [-11.353, -27.243, 111.703, -15.342, -83.794, 50.692]
  Call Extruder(0.135)
  MoveL 4014 to (501.82, 492.3, 8.3) mm, rotated rx 0 ry 90 rz 0 deg; joints [-11.267, -27.161, 111.149, -15.27, -83.337, 50.809]
  Call Extruder(0.055)
  MoveL 4015 to (501.83, 490.4, 8.3) mm, rotated rx 0 ry 90 rz 0 deg; joints [-11.093, -27.168, 111.194, -15.094, -83.369, 50.781]
  Call Extruder(0.226)
  MoveL 4016 to (509.6, 490.4, 8.3) mm, rotated rx 0 ry 90 rz 0 deg; joints [-10.955, -27.022, 110.261, -14.98, -82.604, 50.972]
  Call Extruder(0.232)
  MoveL 4017 to (509.6, 498.38, 8.3) mm, rotated rx 0 ry 90 rz 0 deg; joints [-11.678, -26.991, 110.069, -15.714, -82.471, 51.099]
  Call Extruder(0.056)
  MoveL 4018 to (507.66, 498.38, 8.3) mm, rotated rx 0 ry 90 rz 0 deg; joints [-11.714, -27.029, 110.302, -15.744, -82.66, 51.05]
  Set speed (120.0 mm/s)
  MoveL 4019 to (507.66, 498.78, 8.3) mm, rotated rx 0 ry 90 rz 0 deg; joints [-11.751, -27.027, 110.292, -15.781, -82.653, 51.056]
  Set speed (1000.0 mm/s)
  MoveL 4020 to (506.96, 498.78, 8.3) mm, rotated rx 0 ry 90 rz 0 deg; joints [-11.764, -27.041, 110.376, -15.791, -82.722, 51.038]
  Set speed (1000.0 mm/s)
  MoveL 4021 to (490.68, 490.68, 8.3) mm, rotated rx 0 ry 90 rz 0 deg; joints [-11.324, -27.357, 112.512, -15.294, -84.463, 50.505]
  Set speed (1000.0 mm/s)
  MoveL 4022 to (490.68, 490.68, 8.4) mm, rotated rx 0 ry 90 rz 0 deg; joints [-11.324, -27.367, 112.517, -15.294, -84.458, 50.506]
  Set speed (30.0 mm/s)
  Call Extruder(0.767)
  MoveL 4023 to (509.32, 509.32, 8.4) mm, rotated rx 0 ry 90 rz 0 deg; joints [-12.669, -26.961, 109.824, -16.721, -82.299, 51.277]
  MoveL 4024 to (509.44, 509.44, 8.4) mm, rotated rx 0 ry 90 rz 0 deg; joints [-12.677, -26.958, 109.805, -16.73, -82.285, 51.282]
  Set speed (120.0 mm/s)
  MoveL 4025 to (508.76, 501.14, 8.4) mm, rotated rx 0 ry 90 rz 0 deg; joints [-11.943, -27.007, 110.106, -15.981, -82.5, 51.124]
  Set speed (30.0 mm/s)
  Call Extruder(0.337)
  MoveL 4026 to (500.58, 509.32, 8.4) mm, rotated rx 0 ry 90 rz 0 deg; joints [-12.847, -27.128, 110.869, -16.869, -83.146, 51.041]
  Set speed (120.0 mm/s)
  MoveL 4027 to (499.42, 509.32, 8.4) mm, rotated rx 0 ry 90 rz 0 deg; joints [-12.872, -27.149, 111.007, -16.889, -83.259, 51.009]
  Set speed (30.0 mm/s)
  Call Extruder(0.360)
  MoveL 4028 to (490.68, 500.58, 8.4) mm, rotated rx 0 ry 90 rz 0 deg; joints [-12.247, -27.334, 112.273, -16.227, -84.278, 50.641]
  Set speed (120.0 mm/s)
  MoveL 4029 to (490.68, 499.42, 8.4) mm, rotated rx 0 ry 90 rz 0 deg; joints [-12.139, -27.338, 112.303, -16.118, -84.299, 50.624]
  Set speed (30.0 mm/s)
  Call Extruder(0.282)
  MoveL 4030 to (497.52, 492.58, 8.4) mm, rotated rx 0 ry 90 rz 0 deg; joints [-11.373, -27.247, 111.661, -15.363, -83.75, 50.706]
  MoveL 4031 to (497.65, 492.45, 8.4) mm, rotated rx 0 ry 90 rz 0 deg; joints [-11.359, -27.245, 111.649, -15.35, -83.74, 50.707]
  Set speed (120.0 mm/s)
  MoveL 4032 to (501.79, 492.32, 8.4) mm, rotated rx 0 ry 90 rz 0 deg; joints [-11.271, -27.172, 111.158, -15.274, -83.335, 50.81]
  Set speed (1000.0 mm/s)
  MoveL 4033 to (502.04, 492.14, 8.4) mm, rotated rx 0 ry 90 rz 0 deg; joints [-11.249, -27.168, 111.133, -15.253, -83.313, 50.813]
  Set speed (30.0 mm/s)
  Call Extruder(0.245)
  MoveL 4034 to (508, 498.1, 8.4) mm, rotated rx 0 ry 90 rz 0 deg; joints [-11.682, -27.034, 110.274, -15.713, -82.627, 51.055]
  MoveL 4035 to (508.12, 498.22, 8.4) mm, rotated rx 0 ry 90 rz 0 deg; joints [-11.691, -27.031, 110.256, -15.722, -82.613, 51.06]
  Set speed (120.0 mm/s)
  MoveL 4036 to (509.32, 490.68, 8.4) mm, rotated rx 0 ry 90 rz 0 deg; joints [-10.985, -27.037, 110.293, -15.01, -82.622, 50.971]
  Set speed (30.0 mm/s)
  Call Extruder(0.767)
  MoveL 4037 to (490.68, 509.32, 8.4) mm, rotated rx 0 ry 90 rz 0 deg; joints [-13.056, -27.301, 112.042, -17.046, -84.108, 50.768]
  MoveL 4038 to (490.56, 509.44, 8.4) mm, rotated rx 0 ry 90 rz 0 deg; joints [-13.07, -27.303, 112.053, -17.06, -84.117, 50.766]
  Set speed (120.0 mm/s)
  MoveL 4039 to (507.59, 498.31, 8.4) mm, rotated rx 0 ry 90 rz 0 deg; joints [-11.709, -27.041, 110.317, -15.738, -82.663, 51.048]
  Set speed (1000.0 mm/s)
  MoveL 4040 to (507.66, 498.38, 8.4) mm, rotated rx 0 ry 90 rz 0 deg; joints [-11.714, -27.04, 110.307, -15.744, -82.655, 51.051]
  Set speed (15.0 mm/s)
  Call Extruder(0.010)
  MoveL 4041 to (507.66, 498.73, 8.4) mm, rotated rx 0 ry 90 rz 0 deg; joints [-11.746, -27.038, 110.298, -15.776, -82.649, 51.057]
  Call Extruder(0.062)
  MoveL 4042 to (507.66, 500.86, 8.4) mm, rotated rx 0 ry 90 rz 0 deg; joints [-11.939, -27.029, 110.244, -15.972, -82.612, 51.091]
  Call Extruder(0.056)
  MoveL 4043 to (509.6, 500.86, 8.4) mm, rotated rx 0 ry 90 rz 0 deg; joints [-11.902, -26.992, 110.011, -15.942, -82.423, 51.141]
  Call Extruder(0.254)
  MoveL 4044 to (509.6, 509.6, 8.4) mm, rotated rx 0 ry 90 rz 0 deg; joints [-12.688, -26.954, 109.782, -16.742, -82.267, 51.289]
  Call Extruder(0.559)
  MoveL 4045 to (490.4, 509.6, 8.4) mm, rotated rx 0 ry 90 rz 0 deg; joints [-13.088, -27.305, 112.067, -17.077, -84.129, 50.764]
  MoveL 4046 to (490.4, 490.4, 8.4) mm, rotated rx 0 ry 90 rz 0 deg; joints [-11.303, -27.373, 112.556, -15.273, -84.491, 50.495]
  Call Extruder(0.199)
  MoveL 4047 to (497.23, 490.4, 8.4) mm, rotated rx 0 ry 90 rz 0 deg; joints [-11.177, -27.259, 111.747, -15.164, -83.816, 50.668]
  Call Extruder(0.055)
  MoveL 4048 to (497.23, 492.3, 8.4) mm, rotated rx 0 ry 90 rz 0 deg; joints [-11.352, -27.253, 111.702, -15.342, -83.783, 50.695]
  Call Extruder(0.132)
  MoveL 4049 to (501.76, 492.3, 8.4) mm, rotated rx 0 ry 90 rz 0 deg; joints [-11.269, -27.173, 111.162, -15.271, -83.338, 50.809]
  Call Extruder(0.055)
  MoveL 4050 to (501.76, 490.4, 8.4) mm, rotated rx 0 ry 90 rz 0 deg; joints [-11.094, -27.179, 111.207, -15.095, -83.37, 50.781]
  Call Extruder(0.228)
  MoveL 4051 to (509.6, 490.4, 8.4) mm, rotated rx 0 ry 90 rz 0 deg; joints [-10.955, -27.033, 110.266, -14.98, -82.599, 50.973]
  Call Extruder(0.232)
  MoveL 4052 to (509.6, 498.38, 8.4) mm, rotated rx 0 ry 90 rz 0 deg; joints [-11.678, -27.002, 110.074, -15.714, -82.466, 51.1]
  Call Extruder(0.046)
  MoveL 4053 to (508.01, 498.38, 8.4) mm, rotated rx 0 ry 90 rz 0 deg; joints [-11.708, -27.033, 110.265, -15.738, -82.621, 51.06]
  Call Extruder(0.007)
  MoveL 4054 to (507.66, 498.38, 8.4) mm, rotated rx 0 ry 90 rz 0 deg; joints [-11.714, -27.04, 110.307, -15.744, -82.655, 51.051]
  Set speed (120.0 mm/s)
  MoveL 4055 to (507.66, 498.73, 8.4) mm, rotated rx 0 ry 90 rz 0 deg; joints [-11.746, -27.038, 110.298, -15.776, -82.649, 51.057]
  Set speed (1000.0 mm/s)
  MoveL 4056 to (507.66, 498.78, 8.4) mm, rotated rx 0 ry 90 rz 0 deg; joints [-11.75, -27.038, 110.297, -15.781, -82.648, 51.058]
  Set speed (1000.0 mm/s)
  MoveL 4057 to (506.96, 498.78, 8.4) mm, rotated rx 0 ry 90 rz 0 deg; joints [-11.764, -27.051, 110.381, -15.791, -82.717, 51.04]
  Set speed (1000.0 mm/s)
  MoveL 4058 to (490.68, 490.68, 8.4) mm, rotated rx 0 ry 90 rz 0 deg; joints [-11.324, -27.367, 112.517, -15.294, -84.458, 50.506]
  Set speed (1000.0 mm/s)
  MoveL 4059 to (490.68, 490.68, 8.5) mm, rotated rx 0 ry 90 rz 0 deg; joints [-11.324, -27.378, 112.522, -15.295, -84.453, 50.508]
  Set speed (30.0 mm/s)
  Call Extruder(0.767)
  MoveL 4060 to (509.32, 509.32, 8.5) mm, rotated rx 0 ry 90 rz 0 deg; joints [-12.669, -26.971, 109.829, -16.721, -82.294, 51.278]
  MoveL 4061 to (509.44, 509.44, 8.5) mm, rotated rx 0 ry 90 rz 0 deg; joints [-12.677, -26.968, 109.811, -16.73, -82.28, 51.284]
  Set speed (120.0 mm/s)
  MoveL 4062 to (508.76, 501.14, 8.5) mm, rotated rx 0 ry 90 rz 0 deg; joints [-11.943, -27.018, 110.111, -15.981, -82.495, 51.125]
  Set speed (30.0 mm/s)
  Call Extruder(0.337)
  MoveL 4063 to (500.58, 509.32, 8.5) mm, rotated rx 0 ry 90 rz 0 deg; joints [-12.847, -27.139, 110.875, -16.869, -83.141, 51.043]
  Set speed (120.0 mm/s)
  MoveL 4064 to (499.42, 509.32, 8.5) mm, rotated rx 0 ry 90 rz 0 deg; joints [-12.872, -27.16, 111.013, -16.889, -83.254, 51.011]
  Set speed (30.0 mm/s)
  Call Extruder(0.360)
  MoveL 4065 to (490.68, 500.58, 8.5) mm, rotated rx 0 ry 90 rz 0 deg; joints [-12.247, -27.345, 112.278, -16.227, -84.272, 50.642]
  Set speed (120.0 mm/s)
  MoveL 4066 to (490.68, 499.42, 8.5) mm, rotated rx 0 ry 90 rz 0 deg; joints [-12.139, -27.349, 112.308, -16.118, -84.294, 50.626]
  Set speed (30.0 mm/s)
  Call Extruder(0.282)
  MoveL 4067 to (497.52, 492.58, 8.5) mm, rotated rx 0 ry 90 rz 0 deg; joints [-11.373, -27.257, 111.666, -15.363, -83.745, 50.707]
  MoveL 4068 to (497.65, 492.45, 8.5) mm, rotated rx 0 ry 90 rz 0 deg; joints [-11.359, -27.256, 111.654, -15.35, -83.735, 50.709]
  Set speed (120.0 mm/s)
  MoveL 4069 to (501.73, 492.32, 8.5) mm, rotated rx 0 ry 90 rz 0 deg; joints [-11.272, -27.184, 111.171, -15.275, -83.336, 50.81]
  Set speed (1000.0 mm/s)
  MoveL 4070 to (501.98, 492.08, 8.5) mm, rotated rx 0 ry 90 rz 0 deg; joints [-11.245, -27.18, 111.147, -15.248, -83.315, 50.812]
  Set speed (30.0 mm/s)
  Call Extruder(0.248)
  MoveL 4071 to (508, 498.1, 8.5) mm, rotated rx 0 ry 90 rz 0 deg; joints [-11.682, -27.045, 110.279, -15.713, -82.622, 51.057]
  MoveL 4072 to (508.12, 498.22, 8.5) mm, rotated rx 0 ry 90 rz 0 deg; joints [-11.691, -27.042, 110.261, -15.722, -82.608, 51.062]
  Set speed (120.0 mm/s)
  MoveL 4073 to (509.32, 490.68, 8.5) mm, rotated rx 0 ry 90 rz 0 deg; joints [-10.985, -27.048, 110.299, -15.01, -82.617, 50.972]
  Set speed (30.0 mm/s)
  Call Extruder(0.767)
  MoveL 4074 to (490.68, 509.32, 8.5) mm, rotated rx 0 ry 90 rz 0 deg; joints [-13.056, -27.312, 112.047, -17.046, -84.103, 50.77]
  MoveL 4075 to (490.56, 509.44, 8.5) mm, rotated rx 0 ry 90 rz 0 deg; joints [-13.07, -27.314, 112.058, -17.06, -84.112, 50.768]
  Set speed (120.0 mm/s)
  MoveL 4076 to (507.59, 498.31, 8.5) mm, rotated rx 0 ry 90 rz 0 deg; joints [-11.709, -27.052, 110.322, -15.738, -82.658, 51.05]
  Set speed (1000.0 mm/s)
  MoveL 4077 to (507.66, 498.38, 8.5) mm, rotated rx 0 ry 90 rz 0 deg; joints [-11.714, -27.05, 110.312, -15.744, -82.65, 51.053]
  Set speed (15.0 mm/s)
  Call Extruder(0.053)
  MoveL 4078 to (507.66, 500.19, 8.5) mm, rotated rx 0 ry 90 rz 0 deg; joints [-11.878, -27.043, 110.267, -15.911, -82.619, 51.082]
  Call Extruder(0.001)
  MoveL 4079 to (507.66, 500.22, 8.5) mm, rotated rx 0 ry 90 rz 0 deg; joints [-11.881, -27.043, 110.266, -15.914, -82.618, 51.082]
  Call Extruder(0.019)
  MoveL 4080 to (507.66, 500.86, 8.5) mm, rotated rx 0 ry 90 rz 0 deg; joints [-11.939, -27.04, 110.25, -15.972, -82.607, 51.093]
  Call Extruder(0.001)
  MoveL 4081 to (507.7, 500.86, 8.5) mm, rotated rx 0 ry 90 rz 0 deg; joints [-11.938, -27.039, 110.246, -15.972, -82.604, 51.094]
  Call Extruder(0.055)
  MoveL 4082 to (509.6, 500.86, 8.5) mm, rotated rx 0 ry 90 rz 0 deg; joints [-11.902, -27.002, 110.017, -15.942, -82.418, 51.143]
  Call Extruder(0.254)
  MoveL 4083 to (509.6, 509.6, 8.5) mm, rotated rx 0 ry 90 rz 0 deg; joints [-12.688, -26.964, 109.787, -16.742, -82.262, 51.291]
  Call Extruder(0.559)
  MoveL 4084 to (490.4, 509.6, 8.5) mm, rotated rx 0 ry 90 rz 0 deg; joints [-13.088, -27.316, 112.072, -17.077, -84.124, 50.766]
  MoveL 4085 to (490.4, 490.4, 8.5) mm, rotated rx 0 ry 90 rz 0 deg; joints [-11.303, -27.384, 112.562, -15.273, -84.486, 50.497]
  Call Extruder(0.200)
  MoveL 4086 to (497.29, 490.4, 8.5) mm, rotated rx 0 ry 90 rz 0 deg; joints [-11.176, -27.269, 111.745, -15.164, -83.806, 50.671]
  Call Extruder(0.055)
  MoveL 4087 to (497.29, 492.3, 8.5) mm, rotated rx 0 ry 90 rz 0 deg; joints [-11.351, -27.262, 111.7, -15.341, -83.773, 50.698]
  Call Extruder(0.128)
  MoveL 4088 to (501.7, 492.3, 8.5) mm, rotated rx 0 ry 90 rz 0 deg; joints [-11.27, -27.184, 111.175, -15.273, -83.339, 50.808]
  Call Extruder(0.055)
  MoveL 4089 to (501.7, 490.4, 8.5) mm, rotated rx 0 ry 90 rz 0 deg; joints [-11.096, -27.191, 111.219, -15.096, -83.371, 50.781]
  Call Extruder(0.230)
  MoveL 4090 to (509.6, 490.4, 8.5) mm, rotated rx 0 ry 90 rz 0 deg; joints [-10.955, -27.043, 110.271, -14.98, -82.594, 50.975]
  Call Extruder(0.232)
  MoveL 4091 to (509.6, 498.38, 8.5) mm, rotated rx 0 ry 90 rz 0 deg; joints [-11.678, -27.012, 110.079, -15.714, -82.461, 51.102]
  Call Extruder(0.056)
  MoveL 4092 to (507.66, 498.38, 8.5) mm, rotated rx 0 ry 90 rz 0 deg; joints [-11.714, -27.05, 110.312, -15.744, -82.65, 51.053]
  Set speed (120.0 mm/s)
  MoveL 4093 to (507.66, 498.78, 8.5) mm, rotated rx 0 ry 90 rz 0 deg; joints [-11.75, -27.048, 110.302, -15.781, -82.643, 51.059]
  Set speed (1000.0 mm/s)
  MoveL 4094 to (506.96, 498.78, 8.5) mm, rotated rx 0 ry 90 rz 0 deg; joints [-11.763, -27.062, 110.386, -15.792, -82.712, 51.041]
  Set speed (1000.0 mm/s)
  MoveL 4095 to (490.68, 490.68, 8.5) mm, rotated rx 0 ry 90 rz 0 deg; joints [-11.324, -27.378, 112.522, -15.295, -84.453, 50.508]
  Set speed (1000.0 mm/s)
  MoveL 4096 to (490.68, 490.68, 8.6) mm, rotated rx 0 ry 90 rz 0 deg; joints [-11.324, -27.389, 112.527, -15.295, -84.448, 50.509]
  Set speed (30.0 mm/s)
  Call Extruder(0.767)
  MoveL 4097 to (509.32, 509.32, 8.6) mm, rotated rx 0 ry 90 rz 0 deg; joints [-12.669, -26.982, 109.834, -16.721, -82.289, 51.28]
  MoveL 4098 to (509.44, 509.44, 8.6) mm, rotated rx 0 ry 90 rz 0 deg; joints [-12.677, -26.979, 109.816, -16.731, -82.275, 51.285]
  Set speed (120.0 mm/s)
  MoveL 4099 to (508.76, 501.13, 8.6) mm, rotated rx 0 ry 90 rz 0 deg; joints [-11.943, -27.028, 110.116, -15.981, -82.49, 51.127]
  Set speed (30.0 mm/s)
  Call Extruder(0.337)
  MoveL 4100 to (500.58, 509.32, 8.6) mm, rotated rx 0 ry 90 rz 0 deg; joints [-12.847, -27.149, 110.88, -16.869, -83.136, 51.044]
  Set speed (120.0 mm/s)
  MoveL 4101 to (499.42, 509.32, 8.6) mm, rotated rx 0 ry 90 rz 0 deg; joints [-12.872, -27.17, 111.018, -16.889, -83.249, 51.012]
  Set speed (30.0 mm/s)
  Call Extruder(0.360)
  MoveL 4102 to (490.68, 500.58, 8.6) mm, rotated rx 0 ry 90 rz 0 deg; joints [-12.247, -27.355, 112.284, -16.227, -84.267, 50.644]
  Set speed (120.0 mm/s)
  MoveL 4103 to (490.68, 499.42, 8.6) mm, rotated rx 0 ry 90 rz 0 deg; joints [-12.139, -27.359, 112.313, -16.118, -84.289, 50.627]
  Set speed (30.0 mm/s)
  Call Extruder(0.282)
  MoveL 4104 to (497.52, 492.58, 8.6) mm, rotated rx 0 ry 90 rz 0 deg; joints [-11.373, -27.268, 111.671, -15.364, -83.74, 50.709]
  MoveL 4105 to (497.65, 492.45, 8.6) mm, rotated rx 0 ry 90 rz 0 deg; joints [-11.359, -27.266, 111.66, -15.35, -83.73, 50.71]
  Set speed (120.0 mm/s)
  MoveL 4106 to (501.66, 492.33, 8.6) mm, rotated rx 0 ry 90 rz 0 deg; joints [-11.273, -27.195, 111.184, -15.276, -83.337, 50.809]
  Set speed (1000.0 mm/s)
  MoveL 4107 to (501.91, 492.01, 8.6) mm, rotated rx 0 ry 90 rz 0 deg; joints [-11.24, -27.192, 111.161, -15.243, -83.317, 50.811]
  Set speed (30.0 mm/s)
  Call Extruder(0.250)
  MoveL 4108 to (507.99, 498.1, 8.6) mm, rotated rx 0 ry 90 rz 0 deg; joints [-11.682, -27.055, 110.284, -15.713, -82.618, 51.058]
  MoveL 4109 to (508.12, 498.22, 8.6) mm, rotated rx 0 ry 90 rz 0 deg; joints [-11.691, -27.052, 110.267, -15.722, -82.603, 51.063]
  Set speed (120.0 mm/s)
  MoveL 4110 to (509.32, 490.68, 8.6) mm, rotated rx 0 ry 90 rz 0 deg; joints [-10.985, -27.058, 110.304, -15.01, -82.612, 50.974]
  Set speed (30.0 mm/s)
  Call Extruder(0.767)
  MoveL 4111 to (490.68, 509.32, 8.6) mm, rotated rx 0 ry 90 rz 0 deg; joints [-13.056, -27.323, 112.052, -17.046, -84.098, 50.771]
  MoveL 4112 to (490.56, 509.44, 8.6) mm, rotated rx 0 ry 90 rz 0 deg; joints [-13.07, -27.324, 112.064, -17.06, -84.107, 50.77]
  Set speed (120.0 mm/s)
  MoveL 4113 to (497.28, 492.37, 8.6) mm, rotated rx 0 ry 90 rz 0 deg; joints [-11.358, -27.273, 111.706, -15.348, -83.768, 50.7]
  Set speed (1000.0 mm/s)
  MoveL 4114 to (497.34, 492.3, 8.6) mm, rotated rx 0 ry 90 rz 0 deg; joints [-11.35, -27.272, 111.699, -15.34, -83.762, 50.7]
  Set speed (15.0 mm/s)
  Call Extruder(0.010)
  MoveL 4115 to (497.7, 492.3, 8.6) mm, rotated rx 0 ry 90 rz 0 deg; joints [-11.344, -27.266, 111.657, -15.335, -83.728, 50.709]
  Call Extruder(0.065)
  MoveL 4116 to (499.94, 492.3, 8.6) mm, rotated rx 0 ry 90 rz 0 deg; joints [-11.302, -27.226, 111.39, -15.3, -83.507, 50.766]
  Call Extruder(0.000)
  MoveL 4117 to (499.94, 492.29, 8.6) mm, rotated rx 0 ry 90 rz 0 deg; joints [-11.301, -27.226, 111.39, -15.299, -83.507, 50.766]
  Call Extruder(0.039)
  MoveL 4118 to (501.29, 492.3, 8.6) mm, rotated rx 0 ry 90 rz 0 deg; joints [-11.277, -27.202, 111.23, -15.279, -83.374, 50.8]
  Call Extruder(0.000)
  MoveL 4119 to (501.29, 492.3, 8.6) mm, rotated rx 0 ry 90 rz 0 deg; joints [-11.278, -27.202, 111.229, -15.279, -83.374, 50.8]
  Call Extruder(0.010)
  MoveL 4120 to (501.64, 492.3, 8.6) mm, rotated rx 0 ry 90 rz 0 deg; joints [-11.271, -27.196, 111.188, -15.274, -83.34, 50.808]
  Call Extruder(0.007)
  MoveL 4121 to (501.64, 491.95, 8.6) mm, rotated rx 0 ry 90 rz 0 deg; joints [-11.239, -27.197, 111.196, -15.241, -83.346, 50.803]
  Call Extruder(0.000)
  MoveL 4122 to (501.64, 491.95, 8.6) mm, rotated rx 0 ry 90 rz 0 deg; joints [-11.239, -27.197, 111.196, -15.241, -83.346, 50.803]
  Call Extruder(0.045)
  MoveL 4123 to (501.64, 490.4, 8.6) mm, rotated rx 0 ry 90 rz 0 deg; joints [-11.097, -27.203, 111.232, -15.097, -83.372, 50.781]
  Call Extruder(0.232)
  MoveL 4124 to (509.6, 490.4, 8.6) mm, rotated rx 0 ry 90 rz 0 deg; joints [-10.955, -27.054, 110.277, -14.98, -82.589, 50.976]
  Call Extruder(0.232)
  MoveL 4125 to (509.6, 498.38, 8.6) mm, rotated rx 0 ry 90 rz 0 deg; joints [-11.678, -27.023, 110.084, -15.714, -82.456, 51.103]
  Call Extruder(0.056)
  MoveL 4126 to (507.66, 498.38, 8.6) mm, rotated rx 0 ry 90 rz 0 deg; joints [-11.714, -27.06, 110.317, -15.744, -82.645, 51.054]
  Call Extruder(0.055)
  MoveL 4127 to (507.66, 500.25, 8.6) mm, rotated rx 0 ry 90 rz 0 deg; joints [-11.884, -27.053, 110.27, -15.917, -82.613, 51.084]
  Call Extruder(0.018)
  MoveL 4128 to (507.66, 500.86, 8.6) mm, rotated rx 0 ry 90 rz 0 deg; joints [-11.938, -27.05, 110.255, -15.972, -82.602, 51.094]
  Call Extruder(0.056)
  MoveL 4129 to (509.6, 500.86, 8.6) mm, rotated rx 0 ry 90 rz 0 deg; joints [-11.902, -27.013, 110.022, -15.942, -82.413, 51.144]
  Call Extruder(0.254)
  MoveL 4130 to (509.6, 509.6, 8.6) mm, rotated rx 0 ry 90 rz 0 deg; joints [-12.688, -26.975, 109.793, -16.742, -82.257, 51.292]
  Call Extruder(0.559)
  MoveL 4131 to (490.4, 509.6, 8.6) mm, rotated rx 0 ry 90 rz 0 deg; joints [-13.088, -27.326, 112.078, -17.078, -84.119, 50.768]
  MoveL 4132 to (490.4, 490.4, 8.6) mm, rotated rx 0 ry 90 rz 0 deg; joints [-11.303, -27.394, 112.567, -15.273, -84.48, 50.498]
  Call Extruder(0.202)
  MoveL 4133 to (497.34, 490.4, 8.6) mm, rotated rx 0 ry 90 rz 0 deg; joints [-11.175, -27.279, 111.744, -15.163, -83.795, 50.674]
  Call Extruder(0.045)
  MoveL 4134 to (497.35, 491.95, 8.6) mm, rotated rx 0 ry 90 rz 0 deg; joints [-11.318, -27.273, 111.707, -15.308, -83.768, 50.695]
  Call Extruder(0.007)
  MoveL 4135 to (497.34, 492.3, 8.6) mm, rotated rx 0 ry 90 rz 0 deg; joints [-11.35, -27.272, 111.699, -15.34, -83.762, 50.7]
  Set speed (120.0 mm/s)
  MoveL 4136 to (497.7, 492.3, 8.6) mm, rotated rx 0 ry 90 rz 0 deg; joints [-11.344, -27.266, 111.657, -15.335, -83.728, 50.709]
  Set speed (1000.0 mm/s)
  MoveL 4137 to (497.74, 492.3, 8.6) mm, rotated rx 0 ry 90 rz 0 deg; joints [-11.343, -27.265, 111.651, -15.334, -83.723, 50.71]
  Set speed (1000.0 mm/s)
  MoveL 4138 to (497.75, 493, 8.6) mm, rotated rx 0 ry 90 rz 0 deg; joints [-11.407, -27.263, 111.635, -15.4, -83.711, 50.72]
  Set speed (1000.0 mm/s)
  MoveL 4139 to (490.68, 490.68, 8.6) mm, rotated rx 0 ry 90 rz 0 deg; joints [-11.324, -27.389, 112.527, -15.295, -84.448, 50.509]
  Set speed (1000.0 mm/s)
  MoveL 4140 to (490.68, 490.68, 8.7) mm, rotated rx 0 ry 90 rz 0 deg; joints [-11.324, -27.399, 112.533, -15.295, -84.443, 50.51]
  Set speed (30.0 mm/s)
  Call Extruder(0.767)
  MoveL 4141 to (509.32, 509.32, 8.7) mm, rotated rx 0 ry 90 rz 0 deg; joints [-12.669, -26.992, 109.839, -16.722, -82.284, 51.281]
  MoveL 4142 to (509.44, 509.44, 8.7) mm, rotated rx 0 ry 90 rz 0 deg; joints [-12.677, -26.989, 109.821, -16.731, -82.27, 51.287]
  Set speed (120.0 mm/s)
  MoveL 4143 to (508.76, 501.13, 8.7) mm, rotated rx 0 ry 90 rz 0 deg; joints [-11.943, -27.038, 110.121, -15.981, -82.485, 51.128]
  Set speed (30.0 mm/s)
  Call Extruder(0.337)
  MoveL 4144 to (500.58, 509.32, 8.7) mm, rotated rx 0 ry 90 rz 0 deg; joints [-12.847, -27.16, 110.885, -16.869, -83.131, 51.046]
  Set speed (120.0 mm/s)
  MoveL 4145 to (499.42, 509.32, 8.7) mm, rotated rx 0 ry 90 rz 0 deg; joints [-12.872, -27.181, 111.023, -16.889, -83.244, 51.014]
  Set speed (30.0 mm/s)
  Call Extruder(0.360)
  MoveL 4146 to (490.68, 500.58, 8.7) mm, rotated rx 0 ry 90 rz 0 deg; joints [-12.247, -27.366, 112.289, -16.227, -84.262, 50.645]
  Set speed (120.0 mm/s)
  MoveL 4147 to (490.68, 499.42, 8.7) mm, rotated rx 0 ry 90 rz 0 deg; joints [-12.139, -27.37, 112.318, -16.118, -84.284, 50.629]
  Set speed (30.0 mm/s)
  Call Extruder(0.282)
  MoveL 4148 to (497.52, 492.58, 8.7) mm, rotated rx 0 ry 90 rz 0 deg; joints [-11.373, -27.279, 111.677, -15.364, -83.735, 50.71]
  MoveL 4149 to (497.65, 492.45, 8.7) mm, rotated rx 0 ry 90 rz 0 deg; joints [-11.359, -27.277, 111.665, -15.35, -83.725, 50.712]
  Set speed (120.0 mm/s)
  MoveL 4150 to (501.6, 492.33, 8.7) mm, rotated rx 0 ry 90 rz 0 deg; joints [-11.274, -27.207, 111.197, -15.277, -83.338, 50.809]
  Set speed (1000.0 mm/s)
  MoveL 4151 to (501.85, 491.95, 8.7) mm, rotated rx 0 ry 90 rz 0 deg; joints [-11.235, -27.204, 111.175, -15.239, -83.32, 50.81]
  Set speed (30.0 mm/s)
  Call Extruder(0.253)
  MoveL 4152 to (507.99, 498.09, 8.7) mm, rotated rx 0 ry 90 rz 0 deg; joints [-11.682, -27.066, 110.29, -15.713, -82.613, 51.059]
  MoveL 4153 to (508.12, 498.22, 8.7) mm, rotated rx 0 ry 90 rz 0 deg; joints [-11.691, -27.063, 110.272, -15.722, -82.599, 51.064]
  Set speed (120.0 mm/s)
  MoveL 4154 to (509.32, 490.68, 8.7) mm, rotated rx 0 ry 90 rz 0 deg; joints [-10.985, -27.069, 110.309, -15.01, -82.607, 50.975]
  Set speed (30.0 mm/s)
  Call Extruder(0.767)
  MoveL 4155 to (490.68, 509.32, 8.7) mm, rotated rx 0 ry 90 rz 0 deg; joints [-13.056, -27.333, 112.058, -17.046, -84.093, 50.773]
  MoveL 4156 to (490.56, 509.44, 8.7) mm, rotated rx 0 ry 90 rz 0 deg; joints [-13.07, -27.335, 112.069, -17.06, -84.102, 50.771]
  Set speed (120.0 mm/s)
  MoveL 4157 to (507.59, 498.31, 8.7) mm, rotated rx 0 ry 90 rz 0 deg; joints [-11.709, -27.073, 110.333, -15.739, -82.648, 51.052]
  Set speed (1000.0 mm/s)
  MoveL 4158 to (507.66, 498.38, 8.7) mm, rotated rx 0 ry 90 rz 0 deg; joints [-11.714, -27.071, 110.323, -15.744, -82.64, 51.055]
  Set speed (15.0 mm/s)
  Call Extruder(0.055)
  MoveL 4159 to (507.66, 500.28, 8.7) mm, rotated rx 0 ry 90 rz 0 deg; joints [-11.886, -27.063, 110.275, -15.919, -82.607, 51.086]
  Call Extruder(0.017)
  MoveL 4160 to (507.66, 500.86, 8.7) mm, rotated rx 0 ry 90 rz 0 deg; joints [-11.938, -27.061, 110.26, -15.972, -82.597, 51.096]
  Call Extruder(0.056)
  MoveL 4161 to (509.6, 500.86, 8.7) mm, rotated rx 0 ry 90 rz 0 deg; joints [-11.902, -27.023, 110.027, -15.942, -82.408, 51.145]
  Call Extruder(0.254)
  MoveL 4162 to (509.6, 509.6, 8.7) mm, rotated rx 0 ry 90 rz 0 deg; joints [-12.688, -26.985, 109.798, -16.743, -82.252, 51.294]
  Call Extruder(0.559)
  MoveL 4163 to (490.4, 509.6, 8.7) mm, rotated rx 0 ry 90 rz 0 deg; joints [-13.088, -27.337, 112.083, -17.078, -84.114, 50.769]
  MoveL 4164 to (490.4, 490.4, 8.7) mm, rotated rx 0 ry 90 rz 0 deg; joints [-11.303, -27.405, 112.572, -15.273, -84.475, 50.5]
  Call Extruder(0.204)
  MoveL 4165 to (497.4, 490.4, 8.7) mm, rotated rx 0 ry 90 rz 0 deg; joints [-11.174, -27.288, 111.743, -15.162, -83.784, 50.676]
  Call Extruder(0.055)
  MoveL 4166 to (497.4, 492.3, 8.7) mm, rotated rx 0 ry 90 rz 0 deg; joints [-11.349, -27.282, 111.698, -15.34, -83.752, 50.703]
  Call Extruder(0.121)
  MoveL 4167 to (501.57, 492.3, 8.7) mm, rotated rx 0 ry 90 rz 0 deg; joints [-11.272, -27.208, 111.201, -15.275, -83.341, 50.808]
  Call Extruder(0.055)
  MoveL 4168 to (501.57, 490.4, 8.7) mm, rotated rx 0 ry 90 rz 0 deg; joints [-11.098, -27.214, 111.245, -15.098, -83.373, 50.78]
  Call Extruder(0.234)
  MoveL 4169 to (509.6, 490.4, 8.7) mm, rotated rx 0 ry 90 rz 0 deg; joints [-10.955, -27.064, 110.282, -14.98, -82.583, 50.978]
  Call Extruder(0.232)
  MoveL 4170 to (509.6, 498.38, 8.7) mm, rotated rx 0 ry 90 rz 0 deg; joints [-11.677, -27.033, 110.089, -15.714, -82.451, 51.105]
  Call Extruder(0.056)
  MoveL 4171 to (507.66, 498.38, 8.7) mm, rotated rx 0 ry 90 rz 0 deg; joints [-11.714, -27.071, 110.323, -15.744, -82.64, 51.055]
  Set speed (120.0 mm/s)
  MoveL 4172 to (507.66, 498.77, 8.7) mm, rotated rx 0 ry 90 rz 0 deg; joints [-11.75, -27.069, 110.313, -15.781, -82.633, 51.062]
  Set speed (1000.0 mm/s)
  MoveL 4173 to (506.96, 498.78, 8.7) mm, rotated rx 0 ry 90 rz 0 deg; joints [-11.763, -27.083, 110.397, -15.792, -82.702, 51.044]
  Set speed (1000.0 mm/s)
  MoveL 4174 to (490.68, 490.68, 8.7) mm, rotated rx 0 ry 90 rz 0 deg; joints [-11.324, -27.399, 112.533, -15.295, -84.443, 50.51]
  Set speed (1000.0 mm/s)
  MoveL 4175 to (490.68, 490.68, 8.8) mm, rotated rx 0 ry 90 rz 0 deg; joints [-11.324, -27.41, 112.538, -15.295, -84.437, 50.512]
  Set speed (30.0 mm/s)
  Call Extruder(0.767)
  MoveL 4176 to (509.32, 509.32, 8.8) mm, rotated rx 0 ry 90 rz 0 deg; joints [-12.669, -27.003, 109.844, -16.722, -82.279, 51.283]
  MoveL 4177 to (509.44, 509.44, 8.8) mm, rotated rx 0 ry 90 rz 0 deg; joints [-12.677, -27, 109.826, -16.731, -82.265, 51.288]
  Set speed (120.0 mm/s)
  MoveL 4178 to (508.76, 501.13, 8.8) mm, rotated rx 0 ry 90 rz 0 deg; joints [-11.943, -27.049, 110.126, -15.981, -82.48, 51.13]
  Set speed (30.0 mm/s)
  Call Extruder(0.337)
  MoveL 4179 to (500.58, 509.32, 8.8) mm, rotated rx 0 ry 90 rz 0 deg; joints [-12.847, -27.17, 110.89, -16.869, -83.126, 51.047]
  Set speed (120.0 mm/s)
  MoveL 4180 to (499.42, 509.32, 8.8) mm, rotated rx 0 ry 90 rz 0 deg; joints [-12.872, -27.191, 111.028, -16.89, -83.239, 51.016]
  Set speed (30.0 mm/s)
  Call Extruder(0.360)
  MoveL 4181 to (490.68, 500.58, 8.8) mm, rotated rx 0 ry 90 rz 0 deg; joints [-12.247, -27.377, 112.294, -16.227, -84.257, 50.647]
  Set speed (120.0 mm/s)
  MoveL 4182 to (490.68, 499.42, 8.8) mm, rotated rx 0 ry 90 rz 0 deg; joints [-12.139, -27.381, 112.324, -16.118, -84.279, 50.63]
  Set speed (30.0 mm/s)
  Call Extruder(0.282)
  MoveL 4183 to (497.52, 492.58, 8.8) mm, rotated rx 0 ry 90 rz 0 deg; joints [-11.373, -27.289, 111.682, -15.364, -83.73, 50.712]
  MoveL 4184 to (497.65, 492.45, 8.8) mm, rotated rx 0 ry 90 rz 0 deg; joints [-11.359, -27.287, 111.67, -15.351, -83.72, 50.713]
  Set speed (120.0 mm/s)
  MoveL 4185 to (501.54, 492.33, 8.8) mm, rotated rx 0 ry 90 rz 0 deg; joints [-11.275, -27.219, 111.209, -15.278, -83.339, 50.809]
  Set speed (1000.0 mm/s)
  MoveL 4186 to (501.79, 491.89, 8.8) mm, rotated rx 0 ry 90 rz 0 deg; joints [-11.231, -27.216, 111.19, -15.234, -83.322, 50.809]
  Set speed (30.0 mm/s)
  Call Extruder(0.255)
  MoveL 4187 to (507.99, 498.09, 8.8) mm, rotated rx 0 ry 90 rz 0 deg; joints [-11.682, -27.076, 110.295, -15.713, -82.608, 51.061]
  MoveL 4188 to (508.12, 498.22, 8.8) mm, rotated rx 0 ry 90 rz 0 deg; joints [-11.691, -27.073, 110.277, -15.723, -82.594, 51.066]
  Set speed (120.0 mm/s)
  MoveL 4189 to (509.32, 490.68, 8.8) mm, rotated rx 0 ry 90 rz 0 deg; joints [-10.985, -27.079, 110.314, -15.01, -82.601, 50.976]
  Set speed (30.0 mm/s)
  Call Extruder(0.767)
  MoveL 4190 to (490.68, 509.32, 8.8) mm, rotated rx 0 ry 90 rz 0 deg; joints [-13.056, -27.344, 112.063, -17.046, -84.087, 50.774]
  MoveL 4191 to (490.56, 509.44, 8.8) mm, rotated rx 0 ry 90 rz 0 deg; joints [-13.07, -27.346, 112.074, -17.06, -84.097, 50.773]
  Set speed (120.0 mm/s)
  MoveL 4192 to (507.59, 498.3, 8.8) mm, rotated rx 0 ry 90 rz 0 deg; joints [-11.709, -27.083, 110.338, -15.739, -82.643, 51.054]
  Set speed (1000.0 mm/s)
  MoveL 4193 to (507.66, 498.37, 8.8) mm, rotated rx 0 ry 90 rz 0 deg; joints [-11.714, -27.081, 110.328, -15.744, -82.635, 51.057]
  Set speed (15.0 mm/s)
  Call Extruder(0.056)
  MoveL 4194 to (507.66, 500.31, 8.8) mm, rotated rx 0 ry 90 rz 0 deg; joints [-11.889, -27.074, 110.279, -15.922, -82.602, 51.088]
  Call Extruder(0.016)
  MoveL 4195 to (507.66, 500.85, 8.8) mm, rotated rx 0 ry 90 rz 0 deg; joints [-11.938, -27.071, 110.265, -15.972, -82.592, 51.097]
  Call Extruder(0.056)
  MoveL 4196 to (509.6, 500.86, 8.8) mm, rotated rx 0 ry 90 rz 0 deg; joints [-11.902, -27.034, 110.032, -15.942, -82.403, 51.147]
  Call Extruder(0.254)
  MoveL 4197 to (509.6, 509.6, 8.8) mm, rotated rx 0 ry 90 rz 0 deg; joints [-12.688, -26.996, 109.803, -16.743, -82.247, 51.295]
  Call Extruder(0.559)
  MoveL 4198 to (490.4, 509.6, 8.8) mm, rotated rx 0 ry 90 rz 0 deg; joints [-13.088, -27.348, 112.088, -17.078, -84.109, 50.771]
  MoveL 4199 to (490.4, 490.4, 8.8) mm, rotated rx 0 ry 90 rz 0 deg; joints [-11.303, -27.416, 112.578, -15.273, -84.47, 50.501]
  Call Extruder(0.205)
  MoveL 4200 to (497.46, 490.4, 8.8) mm, rotated rx 0 ry 90 rz 0 deg; joints [-11.173, -27.298, 111.741, -15.161, -83.774, 50.679]
  Call Extruder(0.055)
  MoveL 4201 to (497.46, 492.3, 8.8) mm, rotated rx 0 ry 90 rz 0 deg; joints [-11.348, -27.291, 111.696, -15.339, -83.741, 50.706]
  Call Extruder(0.118)
  MoveL 4202 to (501.51, 492.3, 8.8) mm, rotated rx 0 ry 90 rz 0 deg; joints [-11.273, -27.219, 111.213, -15.276, -83.342, 50.808]
  Call Extruder(0.055)
  MoveL 4203 to (501.51, 490.4, 8.8) mm, rotated rx 0 ry 90 rz 0 deg; joints [-11.099, -27.226, 111.258, -15.099, -83.374, 50.78]
  Call Extruder(0.235)
  MoveL 4204 to (509.6, 490.4, 8.8) mm, rotated rx 0 ry 90 rz 0 deg; joints [-10.955, -27.075, 110.287, -14.981, -82.578, 50.979]
  Call Extruder(0.232)
  MoveL 4205 to (509.6, 498.37, 8.8) mm, rotated rx 0 ry 90 rz 0 deg; joints [-11.677, -27.044, 110.095, -15.714, -82.446, 51.106]
  Call Extruder(0.056)
  MoveL 4206 to (507.66, 498.37, 8.8) mm, rotated rx 0 ry 90 rz 0 deg; joints [-11.714, -27.081, 110.328, -15.744, -82.635, 51.057]
  Set speed (120.0 mm/s)
  MoveL 4207 to (507.66, 498.77, 8.8) mm, rotated rx 0 ry 90 rz 0 deg; joints [-11.75, -27.08, 110.318, -15.781, -82.628, 51.063]
  Set speed (1000.0 mm/s)
  MoveL 4208 to (506.96, 498.77, 8.8) mm, rotated rx 0 ry 90 rz 0 deg; joints [-11.763, -27.093, 110.402, -15.792, -82.697, 51.045]
  Set speed (1000.0 mm/s)
  MoveL 4209 to (490.68, 490.68, 8.8) mm, rotated rx 0 ry 90 rz 0 deg; joints [-11.324, -27.41, 112.538, -15.295, -84.437, 50.512]
  Set speed (1000.0 mm/s)
  MoveL 4210 to (490.68, 490.68, 8.9) mm, rotated rx 0 ry 90 rz 0 deg; joints [-11.324, -27.421, 112.543, -15.295, -84.432, 50.513]
  Set speed (30.0 mm/s)
  Call Extruder(0.767)
  MoveL 4211 to (509.32, 509.32, 8.9) mm, rotated rx 0 ry 90 rz 0 deg; joints [-12.669, -27.013, 109.85, -16.722, -82.274, 51.284]
  MoveL 4212 to (509.44, 509.44, 8.9) mm, rotated rx 0 ry 90 rz 0 deg; joints [-12.677, -27.01, 109.831, -16.731, -82.26, 51.29]
  Set speed (120.0 mm/s)
  MoveL 4213 to (508.77, 501.13, 8.9) mm, rotated rx 0 ry 90 rz 0 deg; joints [-11.942, -27.059, 110.131, -15.981, -82.475, 51.131]
  Set speed (30.0 mm/s)
  Call Extruder(0.337)
  MoveL 4214 to (500.58, 509.32, 8.9) mm, rotated rx 0 ry 90 rz 0 deg; joints [-12.847, -27.181, 110.896, -16.87, -83.121, 51.049]
  Set speed (120.0 mm/s)
  MoveL 4215 to (499.42, 509.32, 8.9) mm, rotated rx 0 ry 90 rz 0 deg; joints [-12.872, -27.202, 111.034, -16.89, -83.233, 51.017]
  Set speed (30.0 mm/s)
  Call Extruder(0.360)
  MoveL 4216 to (490.68, 500.58, 8.9) mm, rotated rx 0 ry 90 rz 0 deg; joints [-12.247, -27.387, 112.299, -16.228, -84.252, 50.648]
  Set speed (120.0 mm/s)
  MoveL 4217 to (490.68, 499.42, 8.9) mm, rotated rx 0 ry 90 rz 0 deg; joints [-12.139, -27.391, 112.329, -16.119, -84.274, 50.632]
  Set speed (30.0 mm/s)
  Call Extruder(0.282)
  MoveL 4218 to (497.52, 492.58, 8.9) mm, rotated rx 0 ry 90 rz 0 deg; joints [-11.373, -27.3, 111.687, -15.364, -83.724, 50.713]
  MoveL 4219 to (497.64, 492.45, 8.9) mm, rotated rx 0 ry 90 rz 0 deg; joints [-11.359, -27.298, 111.675, -15.351, -83.714, 50.714]
  Set speed (120.0 mm/s)
  MoveL 4220 to (501.47, 492.33, 8.9) mm, rotated rx 0 ry 90 rz 0 deg; joints [-11.277, -27.231, 111.222, -15.279, -83.34, 50.809]
  Set speed (1000.0 mm/s)
  MoveL 4221 to (501.72, 491.83, 8.9) mm, rotated rx 0 ry 90 rz 0 deg; joints [-11.226, -27.228, 111.204, -15.229, -83.324, 50.808]
  Set speed (30.0 mm/s)
  Call Extruder(0.258)
  MoveL 4222 to (507.99, 498.09, 8.9) mm, rotated rx 0 ry 90 rz 0 deg; joints [-11.682, -27.087, 110.3, -15.713, -82.603, 51.062]
  MoveL 4223 to (508.12, 498.22, 8.9) mm, rotated rx 0 ry 90 rz 0 deg; joints [-11.691, -27.084, 110.283, -15.723, -82.589, 51.067]
  Set speed (120.0 mm/s)
  MoveL 4224 to (509.32, 490.68, 8.9) mm, rotated rx 0 ry 90 rz 0 deg; joints [-10.985, -27.09, 110.32, -15.01, -82.596, 50.978]
  Set speed (30.0 mm/s)
  Call Extruder(0.767)
  MoveL 4225 to (490.68, 509.32, 8.9) mm, rotated rx 0 ry 90 rz 0 deg; joints [-13.056, -27.355, 112.068, -17.047, -84.082, 50.776]
  MoveL 4226 to (490.56, 509.44, 8.9) mm, rotated rx 0 ry 90 rz 0 deg; joints [-13.07, -27.356, 112.079, -17.06, -84.092, 50.774]
  Set speed (120.0 mm/s)
  MoveL 4227 to (507.59, 498.3, 8.9) mm, rotated rx 0 ry 90 rz 0 deg; joints [-11.709, -27.094, 110.343, -15.739, -82.638, 51.055]
  Set speed (1000.0 mm/s)
  MoveL 4228 to (507.66, 498.37, 8.9) mm, rotated rx 0 ry 90 rz 0 deg; joints [-11.714, -27.092, 110.333, -15.744, -82.63, 51.058]
  Set speed (15.0 mm/s)
  Call Extruder(0.072)
  MoveL 4229 to (507.66, 500.85, 8.9) mm, rotated rx 0 ry 90 rz 0 deg; joints [-11.938, -27.082, 110.271, -15.972, -82.587, 51.098]
  Call Extruder(0.056)
  MoveL 4230 to (509.6, 500.86, 8.9) mm, rotated rx 0 ry 90 rz 0 deg; joints [-11.901, -27.044, 110.038, -15.942, -82.398, 51.148]
  Call Extruder(0.255)
  MoveL 4231 to (509.6, 509.6, 8.9) mm, rotated rx 0 ry 90 rz 0 deg; joints [-12.688, -27.006, 109.808, -16.743, -82.242, 51.297]
  Call Extruder(0.559)
  MoveL 4232 to (490.4, 509.6, 8.9) mm, rotated rx 0 ry 90 rz 0 deg; joints [-13.088, -27.358, 112.093, -17.078, -84.104, 50.772]
  MoveL 4233 to (490.4, 490.4, 8.9) mm, rotated rx 0 ry 90 rz 0 deg; joints [-11.303, -27.426, 112.583, -15.273, -84.465, 50.503]
  Call Extruder(0.207)
  MoveL 4234 to (497.51, 490.4, 8.9) mm, rotated rx 0 ry 90 rz 0 deg; joints [-11.172, -27.307, 111.74, -15.161, -83.763, 50.682]
  Call Extruder(0.055)
  MoveL 4235 to (497.51, 492.3, 8.9) mm, rotated rx 0 ry 90 rz 0 deg; joints [-11.347, -27.301, 111.695, -15.338, -83.73, 50.709]
  Call Extruder(0.114)
  MoveL 4236 to (501.45, 492.3, 8.9) mm, rotated rx 0 ry 90 rz 0 deg; joints [-11.275, -27.231, 111.226, -15.277, -83.343, 50.808]
  Call Extruder(0.055)
  MoveL 4237 to (501.45, 490.4, 8.9) mm, rotated rx 0 ry 90 rz 0 deg; joints [-11.1, -27.238, 111.271, -15.101, -83.375, 50.78]
  Call Extruder(0.237)
  MoveL 4238 to (509.6, 490.4, 8.9) mm, rotated rx 0 ry 90 rz 0 deg; joints [-10.955, -27.085, 110.292, -14.981, -82.573, 50.98]
  Call Extruder(0.232)
  MoveL 4239 to (509.6, 498.37, 8.9) mm, rotated rx 0 ry 90 rz 0 deg; joints [-11.677, -27.054, 110.1, -15.715, -82.441, 51.107]
  Call Extruder(0.056)
  MoveL 4240 to (507.66, 498.37, 8.9) mm, rotated rx 0 ry 90 rz 0 deg; joints [-11.714, -27.092, 110.333, -15.744, -82.63, 51.058]
  Set speed (120.0 mm/s)
  MoveL 4241 to (507.66, 498.77, 8.9) mm, rotated rx 0 ry 90 rz 0 deg; joints [-11.75, -27.09, 110.323, -15.781, -82.623, 51.065]
  Set speed (1000.0 mm/s)
  MoveL 4242 to (506.96, 498.77, 8.9) mm, rotated rx 0 ry 90 rz 0 deg; joints [-11.763, -27.104, 110.407, -15.792, -82.692, 51.047]
  Set speed (1000.0 mm/s)
  MoveL 4243 to (490.68, 490.68, 8.9) mm, rotated rx 0 ry 90 rz 0 deg; joints [-11.324, -27.421, 112.543, -15.295, -84.432, 50.513]
  Set speed (1000.0 mm/s)
  MoveL 4244 to (490.68, 490.68, 9) mm, rotated rx 0 ry 90 rz 0 deg; joints [-11.324, -27.431, 112.549, -15.295, -84.427, 50.515]
  Set speed (30.0 mm/s)
  Call Extruder(0.767)
  MoveL 4245 to (509.32, 509.32, 9) mm, rotated rx 0 ry 90 rz 0 deg; joints [-12.669, -27.024, 109.855, -16.722, -82.269, 51.286]
  MoveL 4246 to (509.44, 509.44, 9) mm, rotated rx 0 ry 90 rz 0 deg; joints [-12.677, -27.021, 109.837, -16.731, -82.255, 51.291]
  Set speed (120.0 mm/s)
  MoveL 4247 to (508.77, 501.13, 9) mm, rotated rx 0 ry 90 rz 0 deg; joints [-11.942, -27.07, 110.136, -15.981, -82.469, 51.133]
  Set speed (30.0 mm/s)
  Call Extruder(0.337)
  MoveL 4248 to (500.58, 509.32, 9) mm, rotated rx 0 ry 90 rz 0 deg; joints [-12.847, -27.191, 110.901, -16.87, -83.116, 51.05]
  Set speed (120.0 mm/s)
  MoveL 4249 to (499.42, 509.32, 9) mm, rotated rx 0 ry 90 rz 0 deg; joints [-12.872, -27.212, 111.039, -16.89, -83.228, 51.019]
  Set speed (30.0 mm/s)
  Call Extruder(0.360)
  MoveL 4250 to (490.68, 500.58, 9) mm, rotated rx 0 ry 90 rz 0 deg; joints [-12.247, -27.398, 112.305, -16.228, -84.247, 50.65]
  Set speed (120.0 mm/s)
  MoveL 4251 to (490.68, 499.42, 9) mm, rotated rx 0 ry 90 rz 0 deg; joints [-12.139, -27.402, 112.334, -16.119, -84.268, 50.633]
  Set speed (30.0 mm/s)
  Call Extruder(0.282)
  MoveL 4252 to (497.52, 492.58, 9) mm, rotated rx 0 ry 90 rz 0 deg; joints [-11.373, -27.31, 111.692, -15.364, -83.719, 50.714]
  MoveL 4253 to (497.64, 492.45, 9) mm, rotated rx 0 ry 90 rz 0 deg; joints [-11.359, -27.309, 111.681, -15.351, -83.709, 50.716]
  Set speed (120.0 mm/s)
  MoveL 4254 to (501.41, 492.32, 9) mm, rotated rx 0 ry 90 rz 0 deg; joints [-11.278, -27.242, 111.235, -15.281, -83.341, 50.809]
  Set speed (1000.0 mm/s)
  MoveL 4255 to (501.66, 491.76, 9) mm, rotated rx 0 ry 90 rz 0 deg; joints [-11.221, -27.24, 111.218, -15.224, -83.326, 50.807]
  Set speed (30.0 mm/s)
  Call Extruder(0.261)
  MoveL 4256 to (507.99, 498.09, 9) mm, rotated rx 0 ry 90 rz 0 deg; joints [-11.682, -27.097, 110.306, -15.713, -82.598, 51.063]
  MoveL 4257 to (508.11, 498.21, 9) mm, rotated rx 0 ry 90 rz 0 deg; joints [-11.691, -27.094, 110.288, -15.723, -82.584, 51.069]
  Set speed (120.0 mm/s)
  MoveL 4258 to (509.32, 490.68, 9) mm, rotated rx 0 ry 90 rz 0 deg; joints [-10.985, -27.1, 110.325, -15.011, -82.591, 50.979]
  Set speed (30.0 mm/s)
  Call Extruder(0.767)
  MoveL 4259 to (490.68, 509.32, 9) mm, rotated rx 0 ry 90 rz 0 deg; joints [-13.056, -27.365, 112.073, -17.047, -84.077, 50.777]
  MoveL 4260 to (490.56, 509.44, 9) mm, rotated rx 0 ry 90 rz 0 deg; joints [-13.07, -27.367, 112.085, -17.061, -84.087, 50.776]
  Set speed (120.0 mm/s)
  MoveL 4261 to (507.59, 498.3, 9) mm, rotated rx 0 ry 90 rz 0 deg; joints [-11.708, -27.104, 110.348, -15.739, -82.633, 51.057]
  Set speed (1000.0 mm/s)
  MoveL 4262 to (507.66, 498.37, 9) mm, rotated rx 0 ry 90 rz 0 deg; joints [-11.714, -27.102, 110.338, -15.744, -82.625, 51.06]
  Set speed (15.0 mm/s)
  Call Extruder(0.058)
  MoveL 4263 to (507.66, 500.37, 9) mm, rotated rx 0 ry 90 rz 0 deg; joints [-11.894, -27.094, 110.288, -15.928, -82.59, 51.092]
  Call Extruder(0.014)
  MoveL 4264 to (507.66, 500.85, 9) mm, rotated rx 0 ry 90 rz 0 deg; joints [-11.938, -27.092, 110.276, -15.973, -82.582, 51.1]
  Call Extruder(0.056)
  MoveL 4265 to (509.6, 500.85, 9) mm, rotated rx 0 ry 90 rz 0 deg; joints [-11.901, -27.055, 110.043, -15.943, -82.393, 51.15]
  Call Extruder(0.255)
  MoveL 4266 to (509.6, 509.6, 9) mm, rotated rx 0 ry 90 rz 0 deg; joints [-12.688, -27.017, 109.813, -16.743, -82.237, 51.298]
  Call Extruder(0.559)
  MoveL 4267 to (490.4, 509.6, 9) mm, rotated rx 0 ry 90 rz 0 deg; joints [-13.088, -27.369, 112.099, -17.078, -84.099, 50.774]
  MoveL 4268 to (490.4, 490.4, 9) mm, rotated rx 0 ry 90 rz 0 deg; joints [-11.303, -27.437, 112.588, -15.273, -84.459, 50.504]
  Call Extruder(0.209)
  MoveL 4269 to (497.57, 490.4, 9) mm, rotated rx 0 ry 90 rz 0 deg; joints [-11.171, -27.317, 111.739, -15.16, -83.752, 50.685]
  Call Extruder(0.055)
  MoveL 4270 to (497.57, 492.3, 9) mm, rotated rx 0 ry 90 rz 0 deg; joints [-11.346, -27.31, 111.694, -15.337, -83.72, 50.712]
  Call Extruder(0.111)
  MoveL 4271 to (501.38, 492.3, 9) mm, rotated rx 0 ry 90 rz 0 deg; joints [-11.276, -27.243, 111.239, -15.278, -83.344, 50.808]
  Call Extruder(0.055)
  MoveL 4272 to (501.38, 490.4, 9) mm, rotated rx 0 ry 90 rz 0 deg; joints [-11.101, -27.25, 111.283, -15.102, -83.376, 50.78]
  Call Extruder(0.239)
  MoveL 4273 to (509.6, 490.4, 9) mm, rotated rx 0 ry 90 rz 0 deg; joints [-10.955, -27.096, 110.297, -14.981, -82.568, 50.982]
  Call Extruder(0.232)
  MoveL 4274 to (509.6, 498.37, 9) mm, rotated rx 0 ry 90 rz 0 deg; joints [-11.677, -27.065, 110.105, -15.715, -82.436, 51.109]
  Call Extruder(0.056)
  MoveL 4275 to (507.66, 498.37, 9) mm, rotated rx 0 ry 90 rz 0 deg; joints [-11.714, -27.102, 110.338, -15.744, -82.625, 51.06]
  Set speed (120.0 mm/s)
  MoveL 4276 to (507.66, 498.77, 9) mm, rotated rx 0 ry 90 rz 0 deg; joints [-11.75, -27.101, 110.328, -15.781, -82.618, 51.066]
  Set speed (1000.0 mm/s)
  MoveL 4277 to (506.96, 498.77, 9) mm, rotated rx 0 ry 90 rz 0 deg; joints [-11.763, -27.114, 110.412, -15.792, -82.686, 51.048]
  Set speed (1000.0 mm/s)
  MoveL 4278 to (490.68, 490.68, 9) mm, rotated rx 0 ry 90 rz 0 deg; joints [-11.324, -27.431, 112.549, -15.295, -84.427, 50.515]
  Set speed (1000.0 mm/s)
  MoveL 4279 to (490.68, 490.68, 9.1) mm, rotated rx 0 ry 90 rz 0 deg; joints [-11.324, -27.442, 112.554, -15.295, -84.422, 50.516]
  Set speed (30.0 mm/s)
  Call Extruder(0.767)
  MoveL 4280 to (509.32, 509.32, 9.1) mm, rotated rx 0 ry 90 rz 0 deg; joints [-12.669, -27.034, 109.86, -16.722, -82.264, 51.287]
  MoveL 4281 to (509.44, 509.44, 9.1) mm, rotated rx 0 ry 90 rz 0 deg; joints [-12.677, -27.031, 109.842, -16.732, -82.25, 51.293]
  Set speed (120.0 mm/s)
  MoveL 4282 to (508.77, 501.13, 9.1) mm, rotated rx 0 ry 90 rz 0 deg; joints [-11.942, -27.08, 110.141, -15.981, -82.464, 51.134]
  Set speed (30.0 mm/s)
  Call Extruder(0.337)
  MoveL 4283 to (500.58, 509.32, 9.1) mm, rotated rx 0 ry 90 rz 0 deg; joints [-12.847, -27.202, 110.906, -16.87, -83.111, 51.052]
  Set speed (120.0 mm/s)
  MoveL 4284 to (499.42, 509.32, 9.1) mm, rotated rx 0 ry 90 rz 0 deg; joints [-12.872, -27.223, 111.044, -16.89, -83.223, 51.02]
  Set speed (30.0 mm/s)
  Call Extruder(0.360)
  MoveL 4285 to (490.68, 500.58, 9.1) mm, rotated rx 0 ry 90 rz 0 deg; joints [-12.247, -27.408, 112.31, -16.228, -84.241, 50.651]
  Set speed (120.0 mm/s)
  MoveL 4286 to (490.68, 499.42, 9.1) mm, rotated rx 0 ry 90 rz 0 deg; joints [-12.139, -27.413, 112.34, -16.119, -84.263, 50.635]
  Set speed (30.0 mm/s)
  Call Extruder(0.282)
  MoveL 4287 to (497.52, 492.58, 9.1) mm, rotated rx 0 ry 90 rz 0 deg; joints [-11.373, -27.321, 111.698, -15.364, -83.714, 50.716]
  MoveL 4288 to (497.65, 492.45, 9.1) mm, rotated rx 0 ry 90 rz 0 deg; joints [-11.359, -27.319, 111.686, -15.351, -83.704, 50.717]
  Set speed (120.0 mm/s)
  MoveL 4289 to (501.35, 492.32, 9.1) mm, rotated rx 0 ry 90 rz 0 deg; joints [-11.279, -27.254, 111.248, -15.282, -83.342, 50.809]
  Set speed (1000.0 mm/s)
  MoveL 4290 to (501.6, 491.7, 9.1) mm, rotated rx 0 ry 90 rz 0 deg; joints [-11.217, -27.252, 111.233, -15.219, -83.328, 50.806]
  Set speed (30.0 mm/s)
  Call Extruder(0.263)
  MoveL 4291 to (507.99, 498.09, 9.1) mm, rotated rx 0 ry 90 rz 0 deg; joints [-11.682, -27.108, 110.311, -15.713, -82.593, 51.065]
  MoveL 4292 to (508.11, 498.21, 9.1) mm, rotated rx 0 ry 90 rz 0 deg; joints [-11.691, -27.105, 110.293, -15.723, -82.579, 51.07]
  Set speed (120.0 mm/s)
  MoveL 4293 to (509.32, 490.68, 9.1) mm, rotated rx 0 ry 90 rz 0 deg; joints [-10.985, -27.111, 110.33, -15.011, -82.586, 50.981]
  Set speed (30.0 mm/s)
  Call Extruder(0.767)
  MoveL 4294 to (490.68, 509.32, 9.1) mm, rotated rx 0 ry 90 rz 0 deg; joints [-13.056, -27.376, 112.079, -17.047, -84.072, 50.779]
  MoveL 4295 to (490.56, 509.44, 9.1) mm, rotated rx 0 ry 90 rz 0 deg; joints [-13.07, -27.377, 112.09, -17.061, -84.082, 50.777]
  Set speed (120.0 mm/s)
  MoveL 4296 to (507.59, 498.3, 9.1) mm, rotated rx 0 ry 90 rz 0 deg; joints [-11.708, -27.115, 110.354, -15.739, -82.628, 51.058]
  Set speed (1000.0 mm/s)
  MoveL 4297 to (507.66, 498.37, 9.1) mm, rotated rx 0 ry 90 rz 0 deg; joints [-11.713, -27.113, 110.343, -15.744, -82.62, 51.061]
  Set speed (15.0 mm/s)
  Call Extruder(0.059)
  MoveL 4298 to (507.66, 500.4, 9.1) mm, rotated rx 0 ry 90 rz 0 deg; joints [-11.897, -27.105, 110.293, -15.931, -82.585, 51.094]
  Call Extruder(0.013)
  MoveL 4299 to (507.66, 500.85, 9.1) mm, rotated rx 0 ry 90 rz 0 deg; joints [-11.938, -27.103, 110.281, -15.973, -82.577, 51.101]
  Call Extruder(0.056)
  MoveL 4300 to (509.6, 500.85, 9.1) mm, rotated rx 0 ry 90 rz 0 deg; joints [-11.901, -27.065, 110.048, -15.943, -82.388, 51.151]
  Call Extruder(0.255)
  MoveL 4301 to (509.6, 509.6, 9.1) mm, rotated rx 0 ry 90 rz 0 deg; joints [-12.688, -27.027, 109.819, -16.743, -82.232, 51.3]
  Call Extruder(0.559)
  MoveL 4302 to (490.4, 509.6, 9.1) mm, rotated rx 0 ry 90 rz 0 deg; joints [-13.088, -27.379, 112.104, -17.078, -84.094, 50.776]
  MoveL 4303 to (490.4, 490.4, 9.1) mm, rotated rx 0 ry 90 rz 0 deg; joints [-11.303, -27.448, 112.593, -15.274, -84.454, 50.505]
  Call Extruder(0.210)
  MoveL 4304 to (497.62, 490.4, 9.1) mm, rotated rx 0 ry 90 rz 0 deg; joints [-11.17, -27.327, 111.737, -15.159, -83.742, 50.688]
  Call Extruder(0.055)
  MoveL 4305 to (497.62, 492.3, 9.1) mm, rotated rx 0 ry 90 rz 0 deg; joints [-11.345, -27.32, 111.692, -15.337, -83.709, 50.715]
  Call Extruder(0.108)
  MoveL 4306 to (501.32, 492.3, 9.1) mm, rotated rx 0 ry 90 rz 0 deg; joints [-11.277, -27.255, 111.252, -15.28, -83.346, 50.807]
  Call Extruder(0.055)
  MoveL 4307 to (501.32, 490.4, 9.1) mm, rotated rx 0 ry 90 rz 0 deg; joints [-11.102, -27.261, 111.296, -15.103, -83.377, 50.78]
  Call Extruder(0.241)
  MoveL 4308 to (509.6, 490.4, 9.1) mm, rotated rx 0 ry 90 rz 0 deg; joints [-10.955, -27.106, 110.303, -14.981, -82.563, 50.983]
  Call Extruder(0.232)
  MoveL 4309 to (509.6, 498.37, 9.1) mm, rotated rx 0 ry 90 rz 0 deg; joints [-11.677, -27.075, 110.11, -15.715, -82.431, 51.11]
  Call Extruder(0.056)
  MoveL 4310 to (507.66, 498.37, 9.1) mm, rotated rx 0 ry 90 rz 0 deg; joints [-11.713, -27.113, 110.343, -15.744, -82.62, 51.061]
  Set speed (120.0 mm/s)
  MoveL 4311 to (507.66, 498.77, 9.1) mm, rotated rx 0 ry 90 rz 0 deg; joints [-11.75, -27.111, 110.334, -15.781, -82.613, 51.068]
  Set speed (1000.0 mm/s)
  MoveL 4312 to (506.96, 498.77, 9.1) mm, rotated rx 0 ry 90 rz 0 deg; joints [-11.763, -27.125, 110.418, -15.792, -82.681, 51.05]
  Set speed (1000.0 mm/s)
  MoveL 4313 to (490.68, 490.68, 9.1) mm, rotated rx 0 ry 90 rz 0 deg; joints [-11.324, -27.442, 112.554, -15.295, -84.422, 50.516]
  Set speed (1000.0 mm/s)
  MoveL 4314 to (490.68, 490.68, 9.2) mm, rotated rx 0 ry 90 rz 0 deg; joints [-11.324, -27.453, 112.559, -15.295, -84.417, 50.518]
  Set speed (30.0 mm/s)
  Call Extruder(0.767)
  MoveL 4315 to (509.32, 509.32, 9.2) mm, rotated rx 0 ry 90 rz 0 deg; joints [-12.669, -27.044, 109.865, -16.723, -82.259, 51.289]
  MoveL 4316 to (509.44, 509.44, 9.2) mm, rotated rx 0 ry 90 rz 0 deg; joints [-12.677, -27.041, 109.847, -16.732, -82.245, 51.294]
  Set speed (120.0 mm/s)
  MoveL 4317 to (508.78, 501.12, 9.2) mm, rotated rx 0 ry 90 rz 0 deg; joints [-11.941, -27.09, 110.145, -15.98, -82.458, 51.136]
  Set speed (30.0 mm/s)
  Call Extruder(0.338)
  MoveL 4318 to (500.58, 509.32, 9.2) mm, rotated rx 0 ry 90 rz 0 deg; joints [-12.847, -27.212, 110.911, -16.87, -83.106, 51.053]
  Set speed (120.0 mm/s)
  MoveL 4319 to (499.42, 509.32, 9.2) mm, rotated rx 0 ry 90 rz 0 deg; joints [-12.872, -27.233, 111.049, -16.89, -83.218, 51.022]
  Set speed (30.0 mm/s)
  Call Extruder(0.360)
  MoveL 4320 to (490.68, 500.58, 9.2) mm, rotated rx 0 ry 90 rz 0 deg; joints [-12.247, -27.419, 112.315, -16.228, -84.236, 50.653]
  Set speed (120.0 mm/s)
  MoveL 4321 to (490.68, 499.42, 9.2) mm, rotated rx 0 ry 90 rz 0 deg; joints [-12.139, -27.423, 112.345, -16.119, -84.258, 50.636]
  Set speed (30.0 mm/s)
  Call Extruder(0.282)
  MoveL 4322 to (497.52, 492.58, 9.2) mm, rotated rx 0 ry 90 rz 0 deg; joints [-11.373, -27.332, 111.703, -15.365, -83.709, 50.717]
  MoveL 4323 to (497.64, 492.45, 9.2) mm, rotated rx 0 ry 90 rz 0 deg; joints [-11.359, -27.33, 111.691, -15.351, -83.699, 50.719]
  Set speed (120.0 mm/s)
  MoveL 4324 to (501.28, 492.33, 9.2) mm, rotated rx 0 ry 90 rz 0 deg; joints [-11.28, -27.266, 111.26, -15.283, -83.343, 50.808]
  Set speed (1000.0 mm/s)
  MoveL 4325 to (501.54, 491.64, 9.2) mm, rotated rx 0 ry 90 rz 0 deg; joints [-11.212, -27.264, 111.247, -15.215, -83.33, 50.805]
  Set speed (30.0 mm/s)
  Call Extruder(0.266)
  MoveL 4326 to (507.99, 498.09, 9.2) mm, rotated rx 0 ry 90 rz 0 deg; joints [-11.682, -27.118, 110.317, -15.714, -82.588, 51.066]
  MoveL 4327 to (508.11, 498.21, 9.2) mm, rotated rx 0 ry 90 rz 0 deg; joints [-11.691, -27.115, 110.299, -15.723, -82.574, 51.071]
  Set speed (120.0 mm/s)
  MoveL 4328 to (509.32, 490.68, 9.2) mm, rotated rx 0 ry 90 rz 0 deg; joints [-10.985, -27.121, 110.335, -15.011, -82.581, 50.982]
  Set speed (30.0 mm/s)
  Call Extruder(0.767)
  MoveL 4329 to (490.68, 509.32, 9.2) mm, rotated rx 0 ry 90 rz 0 deg; joints [-13.056, -27.387, 112.084, -17.047, -84.067, 50.781]
  MoveL 4330 to (490.56, 509.44, 9.2) mm, rotated rx 0 ry 90 rz 0 deg; joints [-13.07, -27.388, 112.095, -17.061, -84.076, 50.779]
  Set speed (120.0 mm/s)
  MoveL 4331 to (507.59, 498.3, 9.2) mm, rotated rx 0 ry 90 rz 0 deg; joints [-11.708, -27.125, 110.359, -15.739, -82.623, 51.06]
  Set speed (1000.0 mm/s)
  MoveL 4332 to (507.66, 498.37, 9.2) mm, rotated rx 0 ry 90 rz 0 deg; joints [-11.713, -27.123, 110.349, -15.744, -82.615, 51.063]
  Set speed (15.0 mm/s)
  Call Extruder(0.071)
  MoveL 4333 to (507.66, 500.82, 9.2) mm, rotated rx 0 ry 90 rz 0 deg; joints [-11.935, -27.113, 110.287, -15.97, -82.572, 51.102]
  Call Extruder(0.056)
  MoveL 4334 to (509.6, 500.85, 9.2) mm, rotated rx 0 ry 90 rz 0 deg; joints [-11.901, -27.075, 110.053, -15.942, -82.383, 51.152]
  Call Extruder(0.255)
  MoveL 4335 to (509.6, 509.6, 9.2) mm, rotated rx 0 ry 90 rz 0 deg; joints [-12.688, -27.038, 109.824, -16.744, -82.226, 51.301]
  Call Extruder(0.559)
  MoveL 4336 to (490.4, 509.6, 9.2) mm, rotated rx 0 ry 90 rz 0 deg; joints [-13.088, -27.39, 112.109, -17.079, -84.088, 50.777]
  MoveL 4337 to (490.4, 490.4, 9.2) mm, rotated rx 0 ry 90 rz 0 deg; joints [-11.303, -27.458, 112.599, -15.274, -84.449, 50.507]
  Call Extruder(0.212)
  MoveL 4338 to (497.68, 490.4, 9.2) mm, rotated rx 0 ry 90 rz 0 deg; joints [-11.169, -27.336, 111.736, -15.159, -83.731, 50.69]
  Call Extruder(0.055)
  MoveL 4339 to (497.68, 492.3, 9.2) mm, rotated rx 0 ry 90 rz 0 deg; joints [-11.344, -27.33, 111.691, -15.336, -83.698, 50.717]
  Call Extruder(0.104)
  MoveL 4340 to (501.26, 492.3, 9.2) mm, rotated rx 0 ry 90 rz 0 deg; joints [-11.278, -27.266, 111.264, -15.281, -83.347, 50.807]
  Call Extruder(0.055)
  MoveL 4341 to (501.26, 490.4, 9.2) mm, rotated rx 0 ry 90 rz 0 deg; joints [-11.104, -27.273, 111.309, -15.104, -83.378, 50.78]
  Call Extruder(0.243)
  MoveL 4342 to (509.6, 490.4, 9.2) mm, rotated rx 0 ry 90 rz 0 deg; joints [-10.955, -27.117, 110.308, -14.981, -82.558, 50.984]
  Call Extruder(0.232)
  MoveL 4343 to (509.6, 498.37, 9.2) mm, rotated rx 0 ry 90 rz 0 deg; joints [-11.677, -27.086, 110.116, -15.715, -82.426, 51.112]
  Call Extruder(0.056)
  MoveL 4344 to (507.66, 498.37, 9.2) mm, rotated rx 0 ry 90 rz 0 deg; joints [-11.713, -27.123, 110.349, -15.744, -82.615, 51.063]
  Set speed (120.0 mm/s)
  MoveL 4345 to (507.66, 498.77, 9.2) mm, rotated rx 0 ry 90 rz 0 deg; joints [-11.75, -27.122, 110.339, -15.781, -82.608, 51.069]
  Set speed (1000.0 mm/s)
  MoveL 4346 to (506.96, 498.77, 9.2) mm, rotated rx 0 ry 90 rz 0 deg; joints [-11.763, -27.135, 110.423, -15.792, -82.676, 51.051]
  Set speed (1000.0 mm/s)
  MoveL 4347 to (490.68, 490.68, 9.2) mm, rotated rx 0 ry 90 rz 0 deg; joints [-11.324, -27.453, 112.559, -15.295, -84.417, 50.518]
  Set speed (1000.0 mm/s)
  MoveL 4348 to (490.68, 490.68, 9.3) mm, rotated rx 0 ry 90 rz 0 deg; joints [-11.324, -27.464, 112.564, -15.296, -84.411, 50.519]
  Set speed (30.0 mm/s)
  Call Extruder(0.767)
  MoveL 4349 to (509.32, 509.32, 9.3) mm, rotated rx 0 ry 90 rz 0 deg; joints [-12.669, -27.055, 109.87, -16.723, -82.254, 51.291]
  MoveL 4350 to (509.44, 509.44, 9.3) mm, rotated rx 0 ry 90 rz 0 deg; joints [-12.677, -27.052, 109.852, -16.732, -82.24, 51.296]
  Set speed (120.0 mm/s)
  MoveL 4351 to (508.77, 501.13, 9.3) mm, rotated rx 0 ry 90 rz 0 deg; joints [-11.942, -27.101, 110.151, -15.981, -82.454, 51.137]
  Set speed (30.0 mm/s)
  Call Extruder(0.337)
  MoveL 4352 to (500.58, 509.32, 9.3) mm, rotated rx 0 ry 90 rz 0 deg; joints [-12.847, -27.223, 110.917, -16.87, -83.101, 51.055]
  Set speed (120.0 mm/s)
  MoveL 4353 to (499.42, 509.32, 9.3) mm, rotated rx 0 ry 90 rz 0 deg; joints [-12.872, -27.244, 111.055, -16.89, -83.213, 51.023]
  Set speed (30.0 mm/s)
  Call Extruder(0.360)
  MoveL 4354 to (490.68, 500.58, 9.3) mm, rotated rx 0 ry 90 rz 0 deg; joints [-12.247, -27.43, 112.321, -16.228, -84.231, 50.654]
  Set speed (120.0 mm/s)
  MoveL 4355 to (490.68, 499.42, 9.3) mm, rotated rx 0 ry 90 rz 0 deg; joints [-12.139, -27.434, 112.35, -16.119, -84.253, 50.638]
  Set speed (30.0 mm/s)
  Call Extruder(0.282)
  MoveL 4356 to (497.52, 492.58, 9.3) mm, rotated rx 0 ry 90 rz 0 deg; joints [-11.373, -27.342, 111.708, -15.365, -83.704, 50.719]
  MoveL 4357 to (497.65, 492.45, 9.3) mm, rotated rx 0 ry 90 rz 0 deg; joints [-11.359, -27.34, 111.696, -15.351, -83.694, 50.72]
  Set speed (120.0 mm/s)
  MoveL 4358 to (501.22, 492.33, 9.3) mm, rotated rx 0 ry 90 rz 0 deg; joints [-11.281, -27.277, 111.273, -15.284, -83.344, 50.808]
  Set speed (1000.0 mm/s)
  MoveL 4359 to (501.47, 491.57, 9.3) mm, rotated rx 0 ry 90 rz 0 deg; joints [-11.207, -27.276, 111.261, -15.21, -83.333, 50.803]
  Set speed (30.0 mm/s)
  Call Extruder(0.267)
  MoveL 4360 to (507.96, 498.07, 9.3) mm, rotated rx 0 ry 90 rz 0 deg; joints [-11.68, -27.129, 110.325, -15.712, -82.585, 51.067]
  MoveL 4361 to (508.09, 498.19, 9.3) mm, rotated rx 0 ry 90 rz 0 deg; joints [-11.689, -27.126, 110.307, -15.721, -82.571, 51.072]
  Set speed (120.0 mm/s)
  MoveL 4362 to (509.32, 490.68, 9.3) mm, rotated rx 0 ry 90 rz 0 deg; joints [-10.985, -27.132, 110.34, -15.011, -82.576, 50.983]
  Set speed (30.0 mm/s)
  Call Extruder(0.767)
  MoveL 4363 to (490.68, 509.32, 9.3) mm, rotated rx 0 ry 90 rz 0 deg; joints [-13.056, -27.397, 112.089, -17.047, -84.062, 50.782]
  MoveL 4364 to (490.56, 509.44, 9.3) mm, rotated rx 0 ry 90 rz 0 deg; joints [-13.07, -27.399, 112.1, -17.061, -84.071, 50.781]
  Set speed (120.0 mm/s)
  MoveL 4365 to (501.26, 492.37, 9.3) mm, rotated rx 0 ry 90 rz 0 deg; joints [-11.284, -27.276, 111.267, -15.287, -83.34, 50.81]
  Set speed (1000.0 mm/s)
  MoveL 4366 to (501.19, 492.3, 9.3) mm, rotated rx 0 ry 90 rz 0 deg; joints [-11.279, -27.278, 111.277, -15.282, -83.348, 50.807]
  Set speed (15.0 mm/s)
  Call Extruder(0.055)
  MoveL 4367 to (501.19, 490.4, 9.3) mm, rotated rx 0 ry 90 rz 0 deg; joints [-11.105, -27.285, 111.322, -15.105, -83.379, 50.779]
  Call Extruder(0.245)
  MoveL 4368 to (509.6, 490.4, 9.3) mm, rotated rx 0 ry 90 rz 0 deg; joints [-10.955, -27.127, 110.313, -14.981, -82.553, 50.986]
  Call Extruder(0.231)
  MoveL 4369 to (509.6, 498.35, 9.3) mm, rotated rx 0 ry 90 rz 0 deg; joints [-11.675, -27.096, 110.121, -15.713, -82.421, 51.113]
  Call Extruder(0.056)
  MoveL 4370 to (507.68, 498.35, 9.3) mm, rotated rx 0 ry 90 rz 0 deg; joints [-11.711, -27.134, 110.353, -15.742, -82.609, 51.064]
  Call Extruder(0.072)
  MoveL 4371 to (507.66, 500.83, 9.3) mm, rotated rx 0 ry 90 rz 0 deg; joints [-11.937, -27.124, 110.292, -15.971, -82.567, 51.104]
  Call Extruder(0.056)
  MoveL 4372 to (509.6, 500.86, 9.3) mm, rotated rx 0 ry 90 rz 0 deg; joints [-11.902, -27.086, 110.058, -15.943, -82.378, 51.154]
  Call Extruder(0.254)
  MoveL 4373 to (509.6, 509.6, 9.3) mm, rotated rx 0 ry 90 rz 0 deg; joints [-12.688, -27.048, 109.829, -16.744, -82.221, 51.303]
  Call Extruder(0.559)
  MoveL 4374 to (490.4, 509.6, 9.3) mm, rotated rx 0 ry 90 rz 0 deg; joints [-13.088, -27.401, 112.114, -17.079, -84.083, 50.779]
  MoveL 4375 to (490.4, 490.4, 9.3) mm, rotated rx 0 ry 90 rz 0 deg; joints [-11.303, -27.469, 112.604, -15.274, -84.444, 50.508]
  Call Extruder(0.213)
  MoveL 4376 to (497.73, 490.4, 9.3) mm, rotated rx 0 ry 90 rz 0 deg; joints [-11.168, -27.346, 111.735, -15.158, -83.72, 50.693]
  Call Extruder(0.055)
  MoveL 4377 to (497.74, 492.3, 9.3) mm, rotated rx 0 ry 90 rz 0 deg; joints [-11.343, -27.339, 111.689, -15.335, -83.688, 50.72]
  Call Extruder(0.101)
  MoveL 4378 to (501.19, 492.3, 9.3) mm, rotated rx 0 ry 90 rz 0 deg; joints [-11.279, -27.278, 111.277, -15.282, -83.348, 50.807]
  Set speed (120.0 mm/s)
  MoveL 4379 to (501.19, 491.9, 9.3) mm, rotated rx 0 ry 90 rz 0 deg; joints [-11.242, -27.279, 111.287, -15.245, -83.354, 50.801]
  Set speed (1000.0 mm/s)
  MoveL 4380 to (501.89, 491.9, 9.3) mm, rotated rx 0 ry 90 rz 0 deg; joints [-11.23, -27.267, 111.203, -15.234, -83.286, 50.819]
  Set speed (1000.0 mm/s)
  MoveL 4381 to (497.71, 492.33, 9.3) mm, rotated rx 0 ry 90 rz 0 deg; joints [-11.346, -27.34, 111.692, -15.338, -83.69, 50.72]
  Set speed (1000.0 mm/s)
  MoveL 4382 to (490.68, 490.68, 9.3) mm, rotated rx 0 ry 90 rz 0 deg; joints [-11.324, -27.464, 112.564, -15.296, -84.411, 50.519]
  Set speed (1000.0 mm/s)
  MoveL 4383 to (490.68, 490.68, 9.4) mm, rotated rx 0 ry 90 rz 0 deg; joints [-11.324, -27.474, 112.57, -15.296, -84.406, 50.521]
  Set speed (30.0 mm/s)
  Call Extruder(0.767)
  MoveL 4384 to (509.32, 509.32, 9.4) mm, rotated rx 0 ry 90 rz 0 deg; joints [-12.669, -27.065, 109.876, -16.723, -82.249, 51.292]
  MoveL 4385 to (509.44, 509.44, 9.4) mm, rotated rx 0 ry 90 rz 0 deg; joints [-12.677, -27.062, 109.857, -16.732, -82.235, 51.297]
  Set speed (120.0 mm/s)
  MoveL 4386 to (508.7, 501.2, 9.4) mm, rotated rx 0 ry 90 rz 0 deg; joints [-11.949, -27.113, 110.163, -15.989, -82.454, 51.138]
  Set speed (30.0 mm/s)
  Call Extruder(0.334)
  MoveL 4387 to (500.58, 509.32, 9.4) mm, rotated rx 0 ry 90 rz 0 deg; joints [-12.847, -27.233, 110.922, -16.87, -83.096, 51.056]
  Set speed (120.0 mm/s)
  MoveL 4388 to (499.42, 509.32, 9.4) mm, rotated rx 0 ry 90 rz 0 deg; joints [-12.872, -27.255, 111.06, -16.891, -83.208, 51.025]
  Set speed (30.0 mm/s)
  Call Extruder(0.360)
  MoveL 4389 to (490.68, 500.58, 9.4) mm, rotated rx 0 ry 90 rz 0 deg; joints [-12.247, -27.44, 112.326, -16.228, -84.226, 50.656]
  Set speed (120.0 mm/s)
  MoveL 4390 to (490.68, 499.42, 9.4) mm, rotated rx 0 ry 90 rz 0 deg; joints [-12.139, -27.445, 112.355, -16.119, -84.248, 50.639]
  Set speed (30.0 mm/s)
  Call Extruder(0.282)
  MoveL 4391 to (497.52, 492.58, 9.4) mm, rotated rx 0 ry 90 rz 0 deg; joints [-11.373, -27.353, 111.713, -15.365, -83.699, 50.72]
  MoveL 4392 to (497.65, 492.45, 9.4) mm, rotated rx 0 ry 90 rz 0 deg; joints [-11.359, -27.351, 111.702, -15.351, -83.689, 50.722]
  Set speed (120.0 mm/s)
  MoveL 4393 to (501.16, 492.33, 9.4) mm, rotated rx 0 ry 90 rz 0 deg; joints [-11.282, -27.289, 111.286, -15.285, -83.345, 50.808]
  Set speed (1000.0 mm/s)
  MoveL 4394 to (501.41, 491.51, 9.4) mm, rotated rx 0 ry 90 rz 0 deg; joints [-11.203, -27.287, 111.275, -15.205, -83.335, 50.802]
  Set speed (30.0 mm/s)
  Call Extruder(0.268)
  MoveL 4395 to (507.91, 498.01, 9.4) mm, rotated rx 0 ry 90 rz 0 deg; joints [-11.676, -27.141, 110.338, -15.708, -82.587, 51.066]
  MoveL 4396 to (508.03, 498.13, 9.4) mm, rotated rx 0 ry 90 rz 0 deg; joints [-11.685, -27.138, 110.32, -15.717, -82.572, 51.071]
  Set speed (120.0 mm/s)
  MoveL 4397 to (509.32, 490.68, 9.4) mm, rotated rx 0 ry 90 rz 0 deg; joints [-10.985, -27.142, 110.346, -15.011, -82.571, 50.985]
  Set speed (30.0 mm/s)
  Call Extruder(0.767)
  MoveL 4398 to (490.68, 509.32, 9.4) mm, rotated rx 0 ry 90 rz 0 deg; joints [-13.056, -27.408, 112.094, -17.047, -84.057, 50.784]
  MoveL 4399 to (490.56, 509.44, 9.4) mm, rotated rx 0 ry 90 rz 0 deg; joints [-13.07, -27.409, 112.106, -17.061, -84.066, 50.782]
  Set speed (120.0 mm/s)
  MoveL 4400 to (507.59, 500.99, 9.4) mm, rotated rx 0 ry 90 rz 0 deg; joints [-11.952, -27.135, 110.302, -15.987, -82.566, 51.106]
  Set speed (1000.0 mm/s)
  MoveL 4401 to (507.66, 500.92, 9.4) mm, rotated rx 0 ry 90 rz 0 deg; joints [-11.944, -27.134, 110.296, -15.979, -82.561, 51.107]
  Set speed (15.0 mm/s)
  Call Extruder(0.056)
  MoveL 4402 to (509.6, 500.92, 9.4) mm, rotated rx 0 ry 90 rz 0 deg; joints [-11.907, -27.096, 110.062, -15.949, -82.372, 51.157]
  Call Extruder(0.253)
  MoveL 4403 to (509.6, 509.6, 9.4) mm, rotated rx 0 ry 90 rz 0 deg; joints [-12.688, -27.058, 109.834, -16.744, -82.216, 51.304]
  Call Extruder(0.559)
  MoveL 4404 to (490.4, 509.6, 9.4) mm, rotated rx 0 ry 90 rz 0 deg; joints [-13.088, -27.411, 112.12, -17.079, -84.078, 50.78]
  MoveL 4405 to (490.4, 490.4, 9.4) mm, rotated rx 0 ry 90 rz 0 deg; joints [-11.303, -27.48, 112.609, -15.274, -84.439, 50.51]
  Call Extruder(0.215)
  MoveL 4406 to (497.79, 490.4, 9.4) mm, rotated rx 0 ry 90 rz 0 deg; joints [-11.167, -27.356, 111.733, -15.157, -83.71, 50.696]
  Call Extruder(0.055)
  MoveL 4407 to (497.79, 492.3, 9.4) mm, rotated rx 0 ry 90 rz 0 deg; joints [-11.342, -27.349, 111.688, -15.335, -83.677, 50.723]
  Call Extruder(0.097)
  MoveL 4408 to (501.13, 492.3, 9.4) mm, rotated rx 0 ry 90 rz 0 deg; joints [-11.28, -27.29, 111.29, -15.283, -83.349, 50.807]
  Call Extruder(0.055)
  MoveL 4409 to (501.13, 490.4, 9.4) mm, rotated rx 0 ry 90 rz 0 deg; joints [-11.106, -27.296, 111.335, -15.106, -83.38, 50.779]
  Call Extruder(0.246)
  MoveL 4410 to (509.6, 490.4, 9.4) mm, rotated rx 0 ry 90 rz 0 deg; joints [-10.955, -27.138, 110.318, -14.982, -82.548, 50.987]
  Call Extruder(0.230)
  MoveL 4411 to (509.6, 498.29, 9.4) mm, rotated rx 0 ry 90 rz 0 deg; joints [-11.669, -27.107, 110.128, -15.708, -82.417, 51.113]
  Call Extruder(0.044)
  MoveL 4412 to (508.1, 498.29, 9.4) mm, rotated rx 0 ry 90 rz 0 deg; joints [-11.698, -27.136, 110.309, -15.731, -82.564, 51.075]
  Call Extruder(0.013)
  MoveL 4413 to (507.66, 498.3, 9.4) mm, rotated rx 0 ry 90 rz 0 deg; joints [-11.707, -27.145, 110.361, -15.738, -82.606, 51.064]
  Call Extruder(0.076)
  MoveL 4414 to (507.66, 500.92, 9.4) mm, rotated rx 0 ry 90 rz 0 deg; joints [-11.944, -27.134, 110.296, -15.979, -82.561, 51.107]
  Set speed (120.0 mm/s)
  MoveL 4415 to (508.06, 500.92, 9.4) mm, rotated rx 0 ry 90 rz 0 deg; joints [-11.936, -27.126, 110.247, -15.973, -82.522, 51.117]
  Set speed (1000.0 mm/s)
  MoveL 4416 to (508.06, 501.61, 9.4) mm, rotated rx 0 ry 90 rz 0 deg; joints [-12, -27.123, 110.23, -16.037, -82.51, 51.128]
  Set speed (1000.0 mm/s)
  MoveL 4417 to (490.68, 490.68, 9.4) mm, rotated rx 0 ry 90 rz 0 deg; joints [-11.324, -27.474, 112.57, -15.296, -84.406, 50.521]
  Set speed (1000.0 mm/s)
  MoveL 4418 to (490.68, 490.68, 9.5) mm, rotated rx 0 ry 90 rz 0 deg; joints [-11.324, -27.485, 112.575, -15.296, -84.401, 50.522]
  Set speed (30.0 mm/s)
  Call Extruder(0.767)
  MoveL 4419 to (509.32, 509.32, 9.5) mm, rotated rx 0 ry 90 rz 0 deg; joints [-12.669, -27.076, 109.881, -16.723, -82.244, 51.294]
  MoveL 4420 to (509.44, 509.44, 9.5) mm, rotated rx 0 ry 90 rz 0 deg; joints [-12.677, -27.073, 109.863, -16.732, -82.23, 51.299]
  Set speed (120.0 mm/s)
  MoveL 4421 to (508.64, 501.25, 9.5) mm, rotated rx 0 ry 90 rz 0 deg; joints [-11.956, -27.124, 110.174, -15.995, -82.454, 51.139]
  Set speed (30.0 mm/s)
  Call Extruder(0.332)
  MoveL 4422 to (500.58, 509.32, 9.5) mm, rotated rx 0 ry 90 rz 0 deg; joints [-12.847, -27.244, 110.927, -16.871, -83.091, 51.058]
  Set speed (120.0 mm/s)
  MoveL 4423 to (499.42, 509.32, 9.5) mm, rotated rx 0 ry 90 rz 0 deg; joints [-12.872, -27.265, 111.065, -16.891, -83.203, 51.026]
  Set speed (30.0 mm/s)
  Call Extruder(0.360)
  MoveL 4424 to (490.68, 500.58, 9.5) mm, rotated rx 0 ry 90 rz 0 deg; joints [-12.247, -27.451, 112.331, -16.229, -84.221, 50.657]
  Set speed (120.0 mm/s)
  MoveL 4425 to (490.68, 499.42, 9.5) mm, rotated rx 0 ry 90 rz 0 deg; joints [-12.139, -27.455, 112.361, -16.12, -84.242, 50.641]
  Set speed (30.0 mm/s)
  Call Extruder(0.283)
  MoveL 4426 to (497.56, 492.53, 9.5) mm, rotated rx 0 ry 90 rz 0 deg; joints [-11.368, -27.363, 111.714, -15.36, -83.69, 50.722]
  MoveL 4427 to (497.69, 492.41, 9.5) mm, rotated rx 0 ry 90 rz 0 deg; joints [-11.354, -27.361, 111.703, -15.347, -83.68, 50.723]
  Set speed (120.0 mm/s)
  MoveL 4428 to (501.09, 492.33, 9.5) mm, rotated rx 0 ry 90 rz 0 deg; joints [-11.284, -27.301, 111.299, -15.286, -83.347, 50.808]
  Set speed (1000.0 mm/s)
  MoveL 4429 to (501.35, 491.45, 9.5) mm, rotated rx 0 ry 90 rz 0 deg; joints [-11.198, -27.299, 111.29, -15.2, -83.337, 50.801]
  Set speed (30.0 mm/s)
  Call Extruder(0.268)
  MoveL 4430 to (507.85, 497.95, 9.5) mm, rotated rx 0 ry 90 rz 0 deg; joints [-11.672, -27.153, 110.352, -15.703, -82.589, 51.065]
  MoveL 4431 to (507.97, 498.07, 9.5) mm, rotated rx 0 ry 90 rz 0 deg; joints [-11.681, -27.15, 110.334, -15.713, -82.574, 51.07]
  Set speed (120.0 mm/s)
  MoveL 4432 to (509.32, 490.68, 9.5) mm, rotated rx 0 ry 90 rz 0 deg; joints [-10.985, -27.153, 110.351, -15.012, -82.566, 50.986]
  Set speed (30.0 mm/s)
  Call Extruder(0.767)
  MoveL 4433 to (490.68, 509.32, 9.5) mm, rotated rx 0 ry 90 rz 0 deg; joints [-13.056, -27.418, 112.1, -17.048, -84.051, 50.785]
  MoveL 4434 to (490.56, 509.44, 9.5) mm, rotated rx 0 ry 90 rz 0 deg; joints [-13.07, -27.42, 112.111, -17.061, -84.061, 50.784]
  Set speed (120.0 mm/s)
  MoveL 4435 to (507.59, 501.04, 9.5) mm, rotated rx 0 ry 90 rz 0 deg; joints [-11.957, -27.145, 110.306, -15.992, -82.56, 51.108]
  Set speed (1000.0 mm/s)
  MoveL 4436 to (507.66, 500.97, 9.5) mm, rotated rx 0 ry 90 rz 0 deg; joints [-11.949, -27.144, 110.299, -15.985, -82.555, 51.109]
  Set speed (15.0 mm/s)
  Call Extruder(0.056)
  MoveL 4437 to (509.6, 500.98, 9.5) mm, rotated rx 0 ry 90 rz 0 deg; joints [-11.912, -27.106, 110.066, -15.955, -82.366, 51.159]
  Call Extruder(0.251)
  MoveL 4438 to (509.6, 509.6, 9.5) mm, rotated rx 0 ry 90 rz 0 deg; joints [-12.688, -27.069, 109.839, -16.744, -82.211, 51.306]
  Call Extruder(0.559)
  MoveL 4439 to (490.4, 509.6, 9.5) mm, rotated rx 0 ry 90 rz 0 deg; joints [-13.088, -27.422, 112.125, -17.079, -84.073, 50.782]
  MoveL 4440 to (490.4, 490.4, 9.5) mm, rotated rx 0 ry 90 rz 0 deg; joints [-11.303, -27.49, 112.614, -15.274, -84.433, 50.511]
  Call Extruder(0.217)
  MoveL 4441 to (497.84, 490.4, 9.5) mm, rotated rx 0 ry 90 rz 0 deg; joints [-11.166, -27.365, 111.732, -15.156, -83.699, 50.699]
  Call Extruder(0.055)
  MoveL 4442 to (497.85, 492.3, 9.5) mm, rotated rx 0 ry 90 rz 0 deg; joints [-11.341, -27.359, 111.687, -15.334, -83.666, 50.726]
